		20:	// Close A
      IF TRUE
      AND THIS^.itfValve_LockA.M_ToHP(tDelay:= T#0MS)
			THEN 
        THIS^.stSeqCtrlGeneral.iInternalSeqStateCase := 30;
			END_IF
      
    30:	// Check if open B
      IF TRUE
			THEN 
        IF THIS^.bOpenChB THEN
          THIS^.stSeqCtrlGeneral.iInternalSeqStateCase := 40;
        ELSE
          THIS^.stSeqCtrlGeneral.iInternalSeqStateCase := 50;
        END_IF
			END_IF

    40:	// Open B
      IF TRUE
      AND THIS^.itfValve_LockB.M_ToWP1(tDelay:= T#0MS)
			THEN 
        THIS^.stSeqCtrlGeneral.iInternalSeqStateCase := 1000;
			END_IF
      
		50:	// Close B
      IF TRUE
      AND THIS^.itfValve_LockB.M_ToHP(tDelay:= T#0MS)
			THEN 
        THIS^.stSeqCtrlGeneral.iInternalSeqStateCase := 1000;
			END_IF
      
    1000: // Exit step
      IF TRUE
			THEN 
				THIS^.stSeqCtrlGeneral.iInternalSeqStateCase := 9999;
			END_IF
      
	ELSE
		THIS^.stSeqCtrlGeneral.eActiveSeqState := E_SEQ_GENERAL.DONE;  
	END_CASE
	THIS^.stSeqCtrlGeneral.strExtraInfo := CONCAT('Internal state: ', TO_STRING(THIS^.stSeqCtrlGeneral.iInternalSeqStateCase));

E_SEQ_GENERAL.DONE:;

E_SEQ_GENERAL.ERROR:;

E_SEQ_GENERAL.TIME_OUT:; 
IF TRUE
AND THIS^.stSeqCtrlGeneral.bTimeOutActiveQuit 
THEN
  THIS^.stSeqCtrlGeneral.strExtraInfo := 'Bitte quittieren und erneut testen';
  IF TRUE
  //AND itfOpMode.P_QUIT
  THEN
    THIS^.stSeqCtrlGeneral.eActiveSeqState := E_SEQ_GENERAL.EXECUTE;
	END_IF
  
END_IF

ELSE
  THIS^.stSeqCtrlGeneral.eActiveSeqState := E_SEQ_GENERAL.ERROR;
END_CASE
END_METHOD

METHOD PRIVATE _m_Seq_PRESSURE_CALIBRATION : E_SEQ_PROCESS
VAR_INPUT
END_VAR
VAR
	ActiveSeq:  STRING;
END_VAR
//THIS^._m_GeneralStepSetting(StepType:=E_STEP_STATE_TYPE.INIT,
ActiveSeq := TO_STRING(THIS^.eSeq);

CASE THIS^.stSeqCtrlGeneral.eActiveSeqState OF
E_SEQ_GENERAL.READY:;

	
E_SEQ_GENERAL.EXECUTE:;
	IF TRUE
	THEN
		THIS^.stSeqCtrlGeneral.eActiveSeqState := E_SEQ_GENERAL.RESET;
	END_IF
  
E_SEQ_GENERAL.RESET:;
	stSeqCtrlGeneral.iInternalSeqStateCase := 0;
	IF TRUE
	THEN
    THIS^.ii := 1;
    FOR THIS^.ii := 1 TO 7 BY 1 DO
      THIS^.listCalibrationTable[THIS^.ii].uiValue := 0;
      THIS^.listCalibrationTable[THIS^.ii].uiPressure := 0;
      THIS^.listCalibrationTable[THIS^.ii].uiState := 0;
		END_FOR
    THIS^.ii := 1;
		THIS^.stSeqCtrlGeneral.eActiveSeqState := E_SEQ_GENERAL.BUSY;
	END_IF
  
E_SEQ_GENERAL.BUSY:;
	CASE THIS^.stSeqCtrlGeneral.iInternalSeqStateCase OF
		0:	// Set work pressure value to XXXX
      IF TRUE
      AND THIS^.itfValve_PressureLimit.M_SetLimit(ePressureType:= E_PRESSURE_TYPE.VALUE, rLimit:= 1000 * THIS^.ii)
			THEN 
        THIS^.listCalibrationTable[THIS^.ii].uiValue := TO_UINT(1000 * THIS^.ii);
        THIS^.listCalibrationTable[THIS^.ii].uiState := 1;
        THIS^.stSeqCtrlGeneral.iInternalSeqStateCase := 10;
			END_IF
      
    10:	// Open A channel
      IF TRUE
      AND THIS^.itfValve_LockA.M_ToWP1(tDelay:= T#10MS)
			THEN 
        IF THIS^.bDoableActing THEN
				  THIS^.stSeqCtrlGeneral.iInternalSeqStateCase := 20;
        ELSE
          THIS^.stSeqCtrlGeneral.iInternalSeqStateCase := 30;
        END_IF
			END_IF
      
    20:	// Open B channel
      IF TRUE
      AND THIS^.itfValve_LockB.M_ToWP1(tDelay:= T#10MS)
			THEN 
				THIS^.stSeqCtrlGeneral.iInternalSeqStateCase := 30;
			END_IF
      
    30: // Move cylinder to WP
      IF TRUE
      AND THIS^.itfValve_CylCtrl.M_ValveCtrl(rSpeedInPercent:= 100, tDelay:= T#10MS)
			THEN 
        THIS^.stSeqCtrlGeneral.iInternalSeqStateCase := 40;
			END_IF
      
    40: // Choice step
      IF TRUE
      THEN
        IF THIS^.ii = 1 THEN
          THIS^.stSeqCtrlGeneral.iInternalSeqStateCase := 50;
        ELSE
          THIS^.stSeqCtrlGeneral.iInternalSeqStateCase := 60;
				END_IF
			END_IF
      
    50: // Delay step (wait for cylinder end position)
      IF TRUE
      AND _m_Delay(DelayTime:= T#30S)
      THEN
        THIS^.stSeqCtrlGeneral.iInternalSeqStateCase := 60;
			END_IF
      
    60: // Delay step (cylinder under load)
      IF TRUE
      AND _m_Delay(DelayTime:= T#5S)
      THEN
        THIS^.stSeqCtrlGeneral.iInternalSeqStateCase := 70;
			END_IF
      
    70: // Save pressure
      IF TRUE
      THEN
        THIS^.listCalibrationTable[THIS^.ii].uiPressure := TO_UINT(THIS^.rCurrentPressureInBar);
        THIS^.listCalibrationTable[THIS^.ii].uiState := 2;
        THIS^.stSeqCtrlGeneral.iInternalSeqStateCase := 80;
			END_IF
      
    80: // Decide step
      IF TRUE
      AND _m_Delay(DelayTime:= T#1S)
      THEN
        IF THIS^.ii >= 7 OR THIS^.ii < 1 THEN
          THIS^.ii := 1;
          THIS^.stSeqCtrlGeneral.iInternalSeqStateCase := 1000;
        ELSE
          THIS^.ii := THIS^.ii + 1;
          THIS^.stSeqCtrlGeneral.iInternalSeqStateCase := 0;
				END_IF
			END_IF
      
    1000: // Stop and exit
      IF TRUE
      AND THIS^.itfValve_PressureLimit.M_SetLimit(ePressureType:= E_PRESSURE_TYPE.VALUE, rLimit:= 0)
      AND THIS^.itfValve_CylCtrl.M_ValveCtrl(rSpeedInPercent:= 0, tDelay:= T#10MS)
      AND THIS^.itfValve_LockA.M_ToHP(tDelay:= T#10MS)
      AND THIS^.itfValve_LockB.M_ToHP(tDelay:= T#10MS)
			THEN 
				THIS^.stSeqCtrlGeneral.iInternalSeqStateCase := 9999;
			END_IF
      
	ELSE
		THIS^.stSeqCtrlGeneral.eActiveSeqState := E_SEQ_GENERAL.DONE;  
	END_CASE
	THIS^.stSeqCtrlGeneral.strExtraInfo := CONCAT('Internal state: ', TO_STRING(THIS^.stSeqCtrlGeneral.iInternalSeqStateCase));

E_SEQ_GENERAL.DONE:;

E_SEQ_GENERAL.ERROR:;

E_SEQ_GENERAL.TIME_OUT:; 
IF TRUE
AND THIS^.stSeqCtrlGeneral.bTimeOutActiveQuit 
THEN
  THIS^.stSeqCtrlGeneral.strExtraInfo := 'Bitte quittieren und erneut testen';
  IF TRUE
  //AND itfOpMode.P_QUIT
  THEN
    THIS^.stSeqCtrlGeneral.eActiveSeqState := E_SEQ_GENERAL.EXECUTE;
	END_IF
  
END_IF

ELSE
  THIS^.stSeqCtrlGeneral.eActiveSeqState := E_SEQ_GENERAL.ERROR;
END_CASE
END_METHOD

METHOD PRIVATE _m_Seq_SET_MAX_POS : E_SEQ_PROCESS
VAR_INPUT
END_VAR
VAR
	ActiveSeq: STRING;
END_VAR
VAR
	
END_VAR
//THIS^._m_GeneralStepSetting(StepType:=E_STEP_STATE_TYPE.INIT,
ActiveSeq := TO_STRING(THIS^.eSeq);

CASE THIS^.stSeqCtrlGeneral.eActiveSeqState OF
E_SEQ_GENERAL.READY:;

	
E_SEQ_GENERAL.EXECUTE:;
	IF TRUE
	THEN
		THIS^.stSeqCtrlGeneral.eActiveSeqState := E_SEQ_GENERAL.RESET;
	END_IF
  
E_SEQ_GENERAL.RESET:;
	stSeqCtrlGeneral.iInternalSeqStateCase := 0;
	IF TRUE
	THEN
		THIS^.stSeqCtrlGeneral.eActiveSeqState := E_SEQ_GENERAL.BUSY;
	END_IF
  
E_SEQ_GENERAL.BUSY:;
	CASE THIS^.stSeqCtrlGeneral.iInternalSeqStateCase OF
		0:	// Set max position
      IF TRUE 
			THEN 
        THIS^.lrPosMax := THIS^.lrCurrentPosAbs / 1000;
        THIS^.stSeqCtrlGeneral.iInternalSeqStateCase := 1000;
			END_IF
      
    1000: // Exit step
      IF TRUE
			THEN 
				THIS^.stSeqCtrlGeneral.iInternalSeqStateCase := 9999;
			END_IF
      
	ELSE
		THIS^.stSeqCtrlGeneral.eActiveSeqState := E_SEQ_GENERAL.DONE;  
	END_CASE
	THIS^.stSeqCtrlGeneral.strExtraInfo := CONCAT('Internal state: ', TO_STRING(THIS^.stSeqCtrlGeneral.iInternalSeqStateCase));

E_SEQ_GENERAL.DONE:;

E_SEQ_GENERAL.ERROR:;

E_SEQ_GENERAL.TIME_OUT:; 
IF TRUE
AND THIS^.stSeqCtrlGeneral.bTimeOutActiveQuit 
THEN
  THIS^.stSeqCtrlGeneral.strExtraInfo := 'Bitte quittieren und erneut testen';
  IF TRUE
  //AND itfOpMode.P_QUIT
  THEN
    THIS^.stSeqCtrlGeneral.eActiveSeqState := E_SEQ_GENERAL.EXECUTE;
	END_IF
  
END_IF

ELSE
  THIS^.stSeqCtrlGeneral.eActiveSeqState := E_SEQ_GENERAL.ERROR;
END_CASE
END_METHOD

METHOD PRIVATE _m_Seq_SET_WORK_PRESSURE : E_SEQ_PROCESS
VAR_INPUT
END_VAR
VAR
	ActiveSeq: STRING;
END_VAR
VAR
	
END_VAR
//THIS^._m_GeneralStepSetting(StepType:=E_STEP_STATE_TYPE.INIT,
ActiveSeq := TO_STRING(THIS^.eSeq);

CASE THIS^.stSeqCtrlGeneral.eActiveSeqState OF
E_SEQ_GENERAL.READY:;

	
E_SEQ_GENERAL.EXECUTE:;
	IF TRUE
	THEN
		THIS^.stSeqCtrlGeneral.eActiveSeqState := E_SEQ_GENERAL.RESET;
	END_IF
  
E_SEQ_GENERAL.RESET:;
	stSeqCtrlGeneral.iInternalSeqStateCase := 0;
	IF TRUE
	THEN
		THIS^.stSeqCtrlGeneral.eActiveSeqState := E_SEQ_GENERAL.BUSY;
	END_IF
  
E_SEQ_GENERAL.BUSY:;
	CASE THIS^.stSeqCtrlGeneral.iInternalSeqStateCase OF
		0:	// Set work pressure
      IF TRUE
      AND THIS^.itfValve_PressureLimit.M_SetLimit(ePressureType:= E_PRESSURE_TYPE.VALUE, rLimit:= TO_REAL(THIS^.iTargetPressureAsValueA))
			THEN 
        THIS^.stSeqCtrlGeneral.iInternalSeqStateCase := 1000;
			END_IF
      
    1000: // Exit step
      IF TRUE
			THEN 
				THIS^.stSeqCtrlGeneral.iInternalSeqStateCase := 9999;
			END_IF
      
	ELSE
		THIS^.stSeqCtrlGeneral.eActiveSeqState := E_SEQ_GENERAL.DONE;  
	END_CASE
	THIS^.stSeqCtrlGeneral.strExtraInfo := CONCAT('Internal state: ', TO_STRING(THIS^.stSeqCtrlGeneral.iInternalSeqStateCase));

E_SEQ_GENERAL.DONE:;

E_SEQ_GENERAL.ERROR:;

E_SEQ_GENERAL.TIME_OUT:; 
IF TRUE
AND THIS^.stSeqCtrlGeneral.bTimeOutActiveQuit 
THEN
  THIS^.stSeqCtrlGeneral.strExtraInfo := 'Bitte quittieren und erneut testen';
  IF TRUE
  //AND itfOpMode.P_QUIT
  THEN
    THIS^.stSeqCtrlGeneral.eActiveSeqState := E_SEQ_GENERAL.EXECUTE;
	END_IF
  
END_IF

ELSE
  THIS^.stSeqCtrlGeneral.eActiveSeqState := E_SEQ_GENERAL.ERROR;
END_CASE
END_METHOD

METHOD PRIVATE _m_Seq_SET_WORK_PRESSURE_ZERO : E_SEQ_PROCESS
VAR_INPUT
END_VAR
VAR
	ActiveSeq: STRING;
END_VAR
VAR
	
END_VAR
//THIS^._m_GeneralStepSetting(StepType:=E_STEP_STATE_TYPE.INIT,
ActiveSeq := TO_STRING(THIS^.eSeq);

CASE THIS^.stSeqCtrlGeneral.eActiveSeqState OF
E_SEQ_GENERAL.READY:;

	
E_SEQ_GENERAL.EXECUTE:;
	IF TRUE
	THEN
		THIS^.stSeqCtrlGeneral.eActiveSeqState := E_SEQ_GENERAL.RESET;
	END_IF
  
E_SEQ_GENERAL.RESET:;
	stSeqCtrlGeneral.iInternalSeqStateCase := 0;
	IF TRUE
	THEN
		THIS^.stSeqCtrlGeneral.eActiveSeqState := E_SEQ_GENERAL.BUSY;
	END_IF
  
E_SEQ_GENERAL.BUSY:;
	CASE THIS^.stSeqCtrlGeneral.iInternalSeqStateCase OF
		0:	// Set work pressure
      IF TRUE
      AND THIS^.itfValve_PressureLimit.M_SetLimit(ePressureType:= E_PRESSURE_TYPE.VALUE, rLimit:= 0.0)
			THEN 
        THIS^.stSeqCtrlGeneral.iInternalSeqStateCase := 1000;
			END_IF
      
    1000: // Exit step
      IF TRUE
			THEN 
				THIS^.stSeqCtrlGeneral.iInternalSeqStateCase := 9999;
			END_IF
      
	ELSE
		THIS^.stSeqCtrlGeneral.eActiveSeqState := E_SEQ_GENERAL.DONE;  
	END_CASE
	THIS^.stSeqCtrlGeneral.strExtraInfo := CONCAT('Internal state: ', TO_STRING(THIS^.stSeqCtrlGeneral.iInternalSeqStateCase));

E_SEQ_GENERAL.DONE:;

E_SEQ_GENERAL.ERROR:;

E_SEQ_GENERAL.TIME_OUT:; 
IF TRUE
AND THIS^.stSeqCtrlGeneral.bTimeOutActiveQuit 
THEN
  THIS^.stSeqCtrlGeneral.strExtraInfo := 'Bitte quittieren und erneut testen';
  IF TRUE
  //AND itfOpMode.P_QUIT
  THEN
    THIS^.stSeqCtrlGeneral.eActiveSeqState := E_SEQ_GENERAL.EXECUTE;
	END_IF
  
END_IF

ELSE
  THIS^.stSeqCtrlGeneral.eActiveSeqState := E_SEQ_GENERAL.ERROR;
END_CASE
END_METHOD

METHOD PRIVATE _m_Seq_SET_ZERO_POS : E_SEQ_PROCESS
VAR_INPUT
END_VAR
VAR
	ActiveSeq: STRING;
END_VAR
VAR
	
END_VAR
//THIS^._m_GeneralStepSetting(StepType:=E_STEP_STATE_TYPE.INIT,
ActiveSeq := TO_STRING(THIS^.eSeq);

CASE THIS^.stSeqCtrlGeneral.eActiveSeqState OF
E_SEQ_GENERAL.READY:;

	
E_SEQ_GENERAL.EXECUTE:;
	IF TRUE
	THEN
		THIS^.stSeqCtrlGeneral.eActiveSeqState := E_SEQ_GENERAL.RESET;
	END_IF
  
E_SEQ_GENERAL.RESET:;
	stSeqCtrlGeneral.iInternalSeqStateCase := 0;
	IF TRUE
	THEN
		THIS^.stSeqCtrlGeneral.eActiveSeqState := E_SEQ_GENERAL.BUSY;
	END_IF
  
E_SEQ_GENERAL.BUSY:;
	CASE THIS^.stSeqCtrlGeneral.iInternalSeqStateCase OF
		0:	// Set zero position
      IF TRUE 
			THEN 
        THIS^.lrPosZero := THIS^.lrCurrentPosAbs / 1000;
        THIS^.stSeqCtrlGeneral.iInternalSeqStateCase := 1000;
			END_IF
      
    1000: // Exit step
      IF TRUE
			THEN 
				THIS^.stSeqCtrlGeneral.iInternalSeqStateCase := 9999;
			END_IF
      
	ELSE
		THIS^.stSeqCtrlGeneral.eActiveSeqState := E_SEQ_GENERAL.DONE;  
	END_CASE
	THIS^.stSeqCtrlGeneral.strExtraInfo := CONCAT('Internal state: ', TO_STRING(THIS^.stSeqCtrlGeneral.iInternalSeqStateCase));

E_SEQ_GENERAL.DONE:;

E_SEQ_GENERAL.ERROR:;

E_SEQ_GENERAL.TIME_OUT:; 
IF TRUE
AND THIS^.stSeqCtrlGeneral.bTimeOutActiveQuit 
THEN
  THIS^.stSeqCtrlGeneral.strExtraInfo := 'Bitte quittieren und erneut testen';
  IF TRUE
  //AND itfOpMode.P_QUIT
  THEN
    THIS^.stSeqCtrlGeneral.eActiveSeqState := E_SEQ_GENERAL.EXECUTE;
	END_IF
  
END_IF

ELSE
  THIS^.stSeqCtrlGeneral.eActiveSeqState := E_SEQ_GENERAL.ERROR;
END_CASE
END_METHOD

METHOD PRIVATE _m_Seq_STOP : E_SEQ_PROCESS
VAR_INPUT
END_VAR
VAR
	ActiveSeq: STRING;
END_VAR
VAR
	
END_VAR
//THIS^._m_GeneralStepSetting(StepType:=E_STEP_STATE_TYPE.INIT,
ActiveSeq := TO_STRING(THIS^.eSeq);

CASE THIS^.stSeqCtrlGeneral.eActiveSeqState OF
E_SEQ_GENERAL.READY:;

	
E_SEQ_GENERAL.EXECUTE:;
	IF TRUE
	THEN
    THIS^.bRegulationTrigger := FALSE;
    THIS^.bPressureRegulationTrigger := FALSE;
		THIS^.stSeqCtrlGeneral.eActiveSeqState := E_SEQ_GENERAL.RESET;
	END_IF
  
E_SEQ_GENERAL.RESET:;
	stSeqCtrlGeneral.iInternalSeqStateCase := 0;
	IF TRUE
	THEN
		THIS^.stSeqCtrlGeneral.eActiveSeqState := E_SEQ_GENERAL.BUSY;
	END_IF
  
E_SEQ_GENERAL.BUSY:;
	CASE THIS^.stSeqCtrlGeneral.iInternalSeqStateCase OF
		0: // Switch off valves
      IF TRUE
      AND THIS^.itfValve_CylCtrl.M_ValveCtrl(rSpeedInPercent:= 0, tDelay:= T#0MS)
			THEN 
				THIS^.stSeqCtrlGeneral.iInternalSeqStateCase := 1000;
			END_IF
      
    1000: // Exit step
      IF TRUE
			THEN 
				THIS^.stSeqCtrlGeneral.iInternalSeqStateCase := 9999;
			END_IF
      
	ELSE
		THIS^.stSeqCtrlGeneral.eActiveSeqState := E_SEQ_GENERAL.DONE;  
	END_CASE
	THIS^.stSeqCtrlGeneral.strExtraInfo := CONCAT('Internal state: ', TO_STRING(THIS^.stSeqCtrlGeneral.iInternalSeqStateCase));

E_SEQ_GENERAL.DONE:;

E_SEQ_GENERAL.ERROR:;

E_SEQ_GENERAL.TIME_OUT:; 
IF TRUE
AND THIS^.stSeqCtrlGeneral.bTimeOutActiveQuit 
THEN
  THIS^.stSeqCtrlGeneral.strExtraInfo := 'Bitte quittieren und erneut testen';
  IF TRUE
  //AND itfOpMode.P_QUIT
  THEN
    THIS^.stSeqCtrlGeneral.eActiveSeqState := E_SEQ_GENERAL.EXECUTE;
	END_IF
  
END_IF

ELSE
  THIS^.stSeqCtrlGeneral.eActiveSeqState := E_SEQ_GENERAL.ERROR;
END_CASE
END_METHOD

METHOD PRIVATE _m_Seq_STOP_AND_LOCK : E_SEQ_PROCESS
VAR_INPUT
END_VAR
VAR
	ActiveSeq: STRING;
END_VAR
VAR
	
END_VAR
//THIS^._m_GeneralStepSetting(StepType:=E_STEP_STATE_TYPE.INIT,
ActiveSeq := TO_STRING(THIS^.eSeq);

CASE THIS^.stSeqCtrlGeneral.eActiveSeqState OF
E_SEQ_GENERAL.READY:;

	
E_SEQ_GENERAL.EXECUTE:;
	IF TRUE
	THEN
    THIS^.bRegulationTrigger := FALSE;
    THIS^.bPressureRegulationTrigger := FALSE;
		THIS^.stSeqCtrlGeneral.eActiveSeqState := E_SEQ_GENERAL.RESET;
	END_IF
  
E_SEQ_GENERAL.RESET:;
	stSeqCtrlGeneral.iInternalSeqStateCase := 0;
	IF TRUE
	THEN
		THIS^.stSeqCtrlGeneral.eActiveSeqState := E_SEQ_GENERAL.BUSY;
	END_IF
  
E_SEQ_GENERAL.BUSY:;
	CASE THIS^.stSeqCtrlGeneral.iInternalSeqStateCase OF
		0: // Switch off valves
      IF TRUE
      AND THIS^.itfValve_CylCtrl.M_ValveCtrl(rSpeedInPercent:= 0, tDelay:= T#0MS)
      AND THIS^.itfValve_LockA.M_ToHP(tDelay:= T#0MS)
      AND THIS^.itfValve_LockB.M_ToHP(tDelay:= T#0MS)
			THEN 
				THIS^.stSeqCtrlGeneral.iInternalSeqStateCase := 1000;
			END_IF
      
    1000: // Exit step
      IF TRUE
			THEN 
				THIS^.stSeqCtrlGeneral.iInternalSeqStateCase := 9999;
			END_IF
      
	ELSE
		THIS^.stSeqCtrlGeneral.eActiveSeqState := E_SEQ_GENERAL.DONE;  
	END_CASE
	THIS^.stSeqCtrlGeneral.strExtraInfo := CONCAT('Internal state: ', TO_STRING(THIS^.stSeqCtrlGeneral.iInternalSeqStateCase));

E_SEQ_GENERAL.DONE:;

E_SEQ_GENERAL.ERROR:;

E_SEQ_GENERAL.TIME_OUT:; 
IF TRUE
AND THIS^.stSeqCtrlGeneral.bTimeOutActiveQuit 
THEN
  THIS^.stSeqCtrlGeneral.strExtraInfo := 'Bitte quittieren und erneut testen';
  IF TRUE
  //AND itfOpMode.P_QUIT
  THEN
    THIS^.stSeqCtrlGeneral.eActiveSeqState := E_SEQ_GENERAL.EXECUTE;
	END_IF
  
END_IF

ELSE
  THIS^.stSeqCtrlGeneral.eActiveSeqState := E_SEQ_GENERAL.ERROR;
END_CASE
END_METHOD

METHOD PRIVATE _m_Seq_TO_HP : E_SEQ_PROCESS
VAR_INPUT
END_VAR
VAR
	ActiveSeq: STRING;
END_VAR
//THIS^._m_GeneralStepSetting(StepType:=E_STEP_STATE_TYPE.INIT,
ActiveSeq := TO_STRING(THIS^.eSeq);

CASE THIS^.stSeqCtrlGeneral.eActiveSeqState OF
E_SEQ_GENERAL.READY:;

	
E_SEQ_GENERAL.EXECUTE:;
	IF TRUE
	THEN
    THIS^.bRegulationTrigger := FALSE;
    THIS^.bPressureRegulationTrigger := FALSE;
		THIS^.stSeqCtrlGeneral.eActiveSeqState := E_SEQ_GENERAL.RESET;
	END_IF
  
E_SEQ_GENERAL.RESET:;
	stSeqCtrlGeneral.iInternalSeqStateCase := 0;
	IF TRUE
	THEN
		THIS^.stSeqCtrlGeneral.eActiveSeqState := E_SEQ_GENERAL.BUSY;
	END_IF
  
E_SEQ_GENERAL.BUSY:;
	CASE THIS^.stSeqCtrlGeneral.iInternalSeqStateCase OF
		0:	// Set work pressure
      IF TRUE
      AND THIS^.itfValve_PressureLimit.M_SetLimit(ePressureType:= E_PRESSURE_TYPE.VALUE, rLimit:= TO_REAL(THIS^.iTargetPressureAsValueB))
			THEN 
        THIS^.stSeqCtrlGeneral.iInternalSeqStateCase := 10;
			END_IF
    
    10:	// Switch on lock A valve
      IF TRUE
      AND THIS^.itfValve_LockA.M_ToWP1(tDelay:= T#0MS)
			THEN 
        IF THIS^.bDoableActing THEN
          THIS^.stSeqCtrlGeneral.iInternalSeqStateCase := 20;
        ELSE
          THIS^.stSeqCtrlGeneral.iInternalSeqStateCase := 30;
        END_IF
			END_IF
      
    20:	// Switch on lock B valve
      IF TRUE
      AND THIS^.itfValve_LockB.M_ToWP1(tDelay:= T#0MS)
			THEN 
        THIS^.stSeqCtrlGeneral.iInternalSeqStateCase := 30;
			END_IF
      
    30:	// Set valve control
      IF TRUE
      AND THIS^.itfValve_CylCtrl.M_ValveCtrl(rSpeedInPercent:= THIS^.rSpeedInPercentToSet, tDelay:= T#0MS)
			THEN 
        THIS^.stSeqCtrlGeneral.iInternalSeqStateCase := 1000;
			END_IF
      
    1000: // Exit step
      IF TRUE
			THEN 
				THIS^.stSeqCtrlGeneral.iInternalSeqStateCase := 9999;
			END_IF
      
	ELSE
		THIS^.stSeqCtrlGeneral.eActiveSeqState := E_SEQ_GENERAL.DONE;  
	END_CASE
	THIS^.stSeqCtrlGeneral.strExtraInfo := CONCAT('Internal state: ', TO_STRING(THIS^.stSeqCtrlGeneral.iInternalSeqStateCase));

E_SEQ_GENERAL.DONE:;
  THIS^.bRegulationTrigger := THIS^.bRegulation;
  THIS^.bPressureRegulationTrigger := THIS^.bPressureRegulation;

E_SEQ_GENERAL.ERROR:;

E_SEQ_GENERAL.TIME_OUT:; 
IF TRUE
AND THIS^.stSeqCtrlGeneral.bTimeOutActiveQuit 
THEN
  THIS^.stSeqCtrlGeneral.strExtraInfo := 'Bitte quittieren und erneut testen';
  IF TRUE
  //AND itfOpMode.P_QUIT
  THEN
    THIS^.stSeqCtrlGeneral.eActiveSeqState := E_SEQ_GENERAL.EXECUTE;
	END_IF
  
END_IF

ELSE
  THIS^.stSeqCtrlGeneral.eActiveSeqState := E_SEQ_GENERAL.ERROR;
END_CASE
END_METHOD

METHOD PRIVATE _m_Seq_TO_SET_POS : E_SEQ_PROCESS
VAR_INPUT
END_VAR
VAR
	ActiveSeq: STRING;
END_VAR
VAR
	
END_VAR
//THIS^._m_GeneralStepSetting(StepType:=E_STEP_STATE_TYPE.INIT,
ActiveSeq := TO_STRING(THIS^.eSeq);

CASE THIS^.stSeqCtrlGeneral.eActiveSeqState OF
E_SEQ_GENERAL.READY:;

	
E_SEQ_GENERAL.EXECUTE:;
	IF TRUE
	THEN
		THIS^.stSeqCtrlGeneral.eActiveSeqState := E_SEQ_GENERAL.RESET;
	END_IF
  
E_SEQ_GENERAL.RESET:;
	stSeqCtrlGeneral.iInternalSeqStateCase := 0;
	IF TRUE
	THEN
		THIS^.stSeqCtrlGeneral.eActiveSeqState := E_SEQ_GENERAL.BUSY;
	END_IF
  
E_SEQ_GENERAL.BUSY:;
	CASE THIS^.stSeqCtrlGeneral.iInternalSeqStateCase OF
		0:	// Switch valves
      IF TRUE
      AND THIS^.itfValve_LockA.M_ToWP1(tDelay:= T#10MS)
      AND THIS^.itfValve_LockB.M_ToWP1(tDelay:= T#10MS)
			THEN 
        IF bStrokeLengthInitialized 
        AND THIS^.lrToSetPos <= THIS^.rStrokeLength 
        AND THIS^.lrToSetPos >= 0.0 
        THEN
          // Set direction
          IF THIS^.lrPos > THIS^.lrToSetPos THEN
            THIS^.rSpeedInPercentToSet := -ABS(THIS^.rSpeedInPercentToSet);
			    END_IF
          THIS^.stSeqCtrlGeneral.iInternalSeqStateCase := 10;
        ELSE
          THIS^.stSeqCtrlGeneral.eActiveSeqState := E_SEQ_GENERAL.ERROR;
				END_IF
			END_IF
      
    10: // Move cylinder to HP and wait for endposition
      IF TRUE
      AND THIS^.itfValve_CylCtrl.M_ValveCtrl(rSpeedInPercent:= THIS^.rSpeedInPercentToSet, tDelay:= T#10MS)
			THEN 
        IF THIS^.lrPos < THIS^.rEndPosTol THEN
				  THIS^.stSeqCtrlGeneral.iInternalSeqStateCase := 20;
        END_IF
			END_IF
      
    20: // Switch off valves
      IF TRUE
      AND THIS^.itfValve_CylCtrl.M_ValveCtrl(rSpeedInPercent:= 0, tDelay:= T#10MS)
			THEN 
				THIS^.stSeqCtrlGeneral.iInternalSeqStateCase := 1000;
			END_IF
      
    1000: // Exit step
      IF TRUE
			THEN 
				THIS^.stSeqCtrlGeneral.iInternalSeqStateCase := 9999;
			END_IF
      
	ELSE
		THIS^.stSeqCtrlGeneral.eActiveSeqState := E_SEQ_GENERAL.DONE;  
	END_CASE
	THIS^.stSeqCtrlGeneral.strExtraInfo := CONCAT('Internal state: ', TO_STRING(THIS^.stSeqCtrlGeneral.iInternalSeqStateCase));

E_SEQ_GENERAL.DONE:;

E_SEQ_GENERAL.ERROR:;

E_SEQ_GENERAL.TIME_OUT:; 
IF TRUE
AND THIS^.stSeqCtrlGeneral.bTimeOutActiveQuit 
THEN
  THIS^.stSeqCtrlGeneral.strExtraInfo := 'Bitte quittieren und erneut testen';
  IF TRUE
  //AND itfOpMode.P_QUIT
  THEN
    THIS^.stSeqCtrlGeneral.eActiveSeqState := E_SEQ_GENERAL.EXECUTE;
	END_IF
  
END_IF

ELSE
  THIS^.stSeqCtrlGeneral.eActiveSeqState := E_SEQ_GENERAL.ERROR;
END_CASE
END_METHOD

METHOD PRIVATE _m_Seq_TO_WP : E_SEQ_PROCESS
VAR_INPUT
END_VAR
VAR
	ActiveSeq: STRING;
END_VAR
VAR
	
END_VAR
//THIS^._m_GeneralStepSetting(StepType:=E_STEP_STATE_TYPE.INIT,
ActiveSeq := TO_STRING(THIS^.eSeq);

CASE THIS^.stSeqCtrlGeneral.eActiveSeqState OF
E_SEQ_GENERAL.READY:;

	
E_SEQ_GENERAL.EXECUTE:;
	IF TRUE
	THEN
    THIS^.bRegulationTrigger := FALSE;
    THIS^.bPressureRegulationTrigger := FALSE;
		THIS^.stSeqCtrlGeneral.eActiveSeqState := E_SEQ_GENERAL.RESET;
	END_IF
  
E_SEQ_GENERAL.RESET:;
	stSeqCtrlGeneral.iInternalSeqStateCase := 0;
	IF TRUE
	THEN
		THIS^.stSeqCtrlGeneral.eActiveSeqState := E_SEQ_GENERAL.BUSY;
	END_IF
  
E_SEQ_GENERAL.BUSY:;
	CASE THIS^.stSeqCtrlGeneral.iInternalSeqStateCase OF
		0:	// Set work pressure
      IF TRUE
      AND THIS^.itfValve_PressureLimit.M_SetLimit(ePressureType:= E_PRESSURE_TYPE.VALUE, rLimit:= TO_REAL(THIS^.iTargetPressureAsValueA))
			THEN 
        THIS^.stSeqCtrlGeneral.iInternalSeqStateCase := 10;
			END_IF

    10:	// Switch on lock A valve
      IF TRUE
      AND THIS^.itfValve_LockA.M_ToWP1(tDelay:= T#0MS)
			THEN 
        IF THIS^.bDoableActing THEN
				  THIS^.stSeqCtrlGeneral.iInternalSeqStateCase := 20;
        ELSE
          THIS^.stSeqCtrlGeneral.iInternalSeqStateCase := 30;
        END_IF
			END_IF
      
    20:	// Switch on lock B valve
      IF TRUE
      AND THIS^.itfValve_LockB.M_ToWP1(tDelay:= T#0MS)
			THEN 
				THIS^.stSeqCtrlGeneral.iInternalSeqStateCase := 30;
			END_IF
      
    30:	// Set valve control
      IF TRUE
      AND THIS^.itfValve_CylCtrl.M_ValveCtrl(rSpeedInPercent:= THIS^.rSpeedInPercentToSet, tDelay:= T#0MS)
			THEN 
				THIS^.stSeqCtrlGeneral.iInternalSeqStateCase := 1000;
			END_IF
      
    1000: // Exit step
      IF TRUE
			THEN 
				THIS^.stSeqCtrlGeneral.iInternalSeqStateCase := 9999;
			END_IF
      
	ELSE
		THIS^.stSeqCtrlGeneral.eActiveSeqState := E_SEQ_GENERAL.DONE;  
	END_CASE
	THIS^.stSeqCtrlGeneral.strExtraInfo := CONCAT('Internal state: ', TO_STRING(THIS^.stSeqCtrlGeneral.iInternalSeqStateCase));

E_SEQ_GENERAL.DONE:;
  THIS^.bRegulationTrigger := THIS^.bRegulation;
  THIS^.bPressureRegulationTrigger := THIS^.bPressureRegulation;
  
E_SEQ_GENERAL.ERROR:;

E_SEQ_GENERAL.TIME_OUT:; 
IF TRUE
AND THIS^.stSeqCtrlGeneral.bTimeOutActiveQuit 
THEN
  THIS^.stSeqCtrlGeneral.strExtraInfo := 'Bitte quittieren und erneut testen';
  IF TRUE
  //AND itfOpMode.P_QUIT
  THEN
    THIS^.stSeqCtrlGeneral.eActiveSeqState := E_SEQ_GENERAL.EXECUTE;
	END_IF
  
END_IF

ELSE
  THIS^.stSeqCtrlGeneral.eActiveSeqState := E_SEQ_GENERAL.ERROR;
END_CASE
END_METHOD

METHOD PRIVATE _m_SequenceManager
VAR_INPUT
END_VAR
IF FALSE
//AND THIS^.eActiveSeqState=DONE 
AND eLastSeq<>eSeq
THEN
	IF THIS^.stSeqCtrlGeneral.eActiveSeqState<>E_SEQ_GENERAL.EXECUTE THEN
		THIS^.stSeqCtrlGeneral.eActiveSeqState:=E_SEQ_GENERAL.READY;
	END_IF
END_IF

eSeq := eNextSeq;

//DelayTimer und TimeOut Timer verwalten
stSeqCtrlGeneral.bActiveStep:=	TRUE
				AND eLastSeq					=	eSeq
				AND stSeqCtrlGeneral.eLastActiveSeqState			=	stSeqCtrlGeneral.eActiveSeqState
				AND	stSeqCtrlGeneral.iLastInternalSeqStateCase	=	stSeqCtrlGeneral.iInternalSeqStateCase
				;
			
IF NOT stSeqCtrlGeneral.bActiveStep THEN
	stSeqCtrlGeneral.bDelayActive:=FALSE;
	stSeqCtrlGeneral.bTimeOutActiveQuit:=FALSE;
	stSeqCtrlGeneral.bTimeOutActiveNoQuit:=FALSE;
  THIS^.stSeqCtrlGeneral.strExtraInfo:='';
END_IF

_m_SaveLastStep();
stSeqCtrlGeneral.tonDelay	(IN:=stSeqCtrlGeneral.bActiveStep AND stSeqCtrlGeneral.bDelayActive, 		PT:=stSeqCtrlGeneral.tDelay);
stSeqCtrlGeneral.tonTimeOut	(IN:=stSeqCtrlGeneral.bActiveStep AND (stSeqCtrlGeneral.bTimeOutActiveNoQuit OR stSeqCtrlGeneral.bTimeOutActiveQuit), 	PT:=stSeqCtrlGeneral.tTimeOut);
stSeqCtrlGeneral.tonStepTime	(IN:= stSeqCtrlGeneral.bActiveStep, PT:= T#24H);

IF stSeqCtrlGeneral.tonTimeOut.Q  THEN
	stSeqCtrlGeneral.eActiveSeqState:=E_SEQ_GENERAL.TIME_OUT;
END_IF

IF stSeqCtrlGeneral.iError<>0 THEN
	eSeq:=E_SEQ_CYLINDER.ERROR_SEQ;
END_IF



eLastSeq					:=	eSeq;
stSeqCtrlGeneral.eLastActiveSeqState			:=	stSeqCtrlGeneral.eActiveSeqState;
stSeqCtrlGeneral.iLastInternalSeqStateCase	:=	stSeqCtrlGeneral.iInternalSeqStateCase;

// Reset set ready state
IF THIS^.stSeqCtrlGeneral.bExitSetReadyState THEN
  THIS^.stSeqCtrlGeneral.bExitSetReadyState := FALSE;
END_IF
END_METHOD

(******************Description****************)
// This function allows variable speed control
(*********************************************)
METHOD PRIVATE _m_SpeedRegulation : BOOL
VAR_INPUT
END_VAR
IF TRUE
AND THIS^.rCurrentSpeedInMmPerS < THIS^.rSpeedInMmPerSToSet 
AND THIS^.rCorrectedSpeedPercent < 100
AND THIS^.bRegulationTrigger
AND NOT THIS^.bRegulationBusy
THEN
  IF ABS(THIS^.rCurrentSpeedInMmPerS - THIS^.rSpeedInMmPerSToSet) > 1 THEN
    //THIS^.rCorrectedSpeedPercent := THIS^.rCorrectedSpeedPercent + 0.25;
    THIS^.rCorrectedSpeedPercent := THIS^.rCorrectedSpeedPercent + ABS((THIS^.rCurrentSpeedInMmPerS - THIS^.rSpeedInMmPerSToSet) * THIS^.rSpeedRegulationFactor);
    THIS^.bCorrectionTrigger := TRUE;
  END_IF
ELSIF TRUE
AND THIS^.rCurrentSpeedInMmPerS > THIS^.rSpeedInMmPerSToSet 
AND THIS^.rCorrectedSpeedPercent > -100
AND THIS^.bRegulationTrigger
AND NOT THIS^.bRegulationBusy
THEN
  IF ABS(THIS^.rCurrentSpeedInMmPerS - THIS^.rSpeedInMmPerSToSet) > 1 THEN
    //THIS^.rCorrectedSpeedPercent := THIS^.rCorrectedSpeedPercent - 0.25;
    THIS^.rCorrectedSpeedPercent := THIS^.rCorrectedSpeedPercent - ABS((THIS^.rCurrentSpeedInMmPerS - THIS^.rSpeedInMmPerSToSet) * THIS^.rSpeedRegulationFactor);
    THIS^.bCorrectionTrigger := TRUE;
  END_IF
END_IF

// Valve value correction
IF THIS^.bCorrectionTrigger THEN
  THIS^.bRegulationBusy:= TRUE;
  CASE THIS^.uiRegulationSeq OF
    0:;
      IF THIS^.itfValve_CylCtrl.M_SetReady() THEN
        THIS^.uiRegulationSeq := 1;
	    END_IF
    1:;
      IF THIS^.itfValve_CylCtrl.M_ValveCtrl(rSpeedInPercent:= THIS^.rCorrectedSpeedPercent, tDelay:= T#0MS) THEN
        THIS^.bCorrectionTrigger := FALSE;
        THIS^.bRegulationBusy := FALSE;
        THIS^.uiRegulationSeq := 0;
	    END_IF
	END_CASE
END_IF
END_METHOD

METHOD PRIVATE _m_TimeOut : BOOL
VAR_INPUT
	bTimeoutActiveToQuit:	BOOL;
	bTimeOutActiveNoQuit:	BOOL;
	tTimeOut:				TIME;	
END_VAR
THIS^.stSeqCtrlGeneral.bTimeOutActiveQuit:=	bTimeoutActiveToQuit;
THIS^.stSeqCtrlGeneral.bTimeOutActiveNoQuit:=	bTimeOutActiveNoQuit;
THIS^.stSeqCtrlGeneral.tTimeOut:=			tTimeOut;
_m_TimeOut:=FALSE;
IF THIS^.stSeqCtrlGeneral.tonTimeOut.Q THEN
	_m_TimeOut:=TRUE;
END_IF
END_METHOD

METHOD FB_init : BOOL
VAR_INPUT
	bInitRetains : BOOL; // if TRUE, the retain variables are initialized (warm start / cold start)
	bInCopyCode : BOOL;  // if TRUE, the instance afterwards gets moved into the copy code (online change)
  
  itfOpMode:											                        I_OP_MODE;
  itfEventLogger:                                         I_EVENT_LOGGER;
  itfOpModeVisu:											                    I_OP_MODE_PAUSE_VISU;
  itfValve_CylCtrl:                                       I_VALVE_X_3_PROP;
  itfValve_LockA:                                         I_VALVE_X_2;
  itfValve_LockB:                                         I_VALVE_X_2;
  itfValve_PressureLimit:                                 I_PRV_PROP; 
  rEndPosTol:                                             REAL;
  /// Volume flow in l/min or dm³/min
  rPumpVolumeFlow:                                        REAL; // Volumenstrom
  /// Pump efficiency factor (0,5-1)
  rPumpEfficiencyFactor:                                  REAL; // Wirkungsgrad
END_VAR
THIS^.itfOpMode := itfOpMode;
THIS^.itfEventLogger := itfEventLogger;
THIS^.itfOpModeVisu := itfOpModeVisu;
THIS^.itfValve_CylCtrl := itfValve_CylCtrl;
THIS^.itfValve_LockA := itfValve_LockA;
THIS^.itfValve_LockB := itfValve_LockB;
THIS^.itfValve_PressureLimit := itfValve_PressureLimit;
THIS^.rEndPosTol := rEndPosTol;
THIS^.rPumpVolumeFlow := rPumpVolumeFlow;
THIS^.rPumpEfficiencyFactor := rPumpEfficiencyFactor;
END_METHOD

METHOD M_OpenLockValves : BOOL
VAR_INPUT
	bOpenChA	: BOOL;
	bOpenChB	: BOOL;
END_VAR
M_OpenLockValves := THIS^.stSeqCtrlGeneral.eActiveSeqState = E_SEQ_GENERAL.DONE;

// Assign input
THIS^.bOpenChA := bOpenChA;
THIS^.bOpenChB := bOpenChB;

// General
IF THIS^.stSeqCtrlGeneral.eActiveSeqState = E_SEQ_GENERAL.READY THEN
  THIS^.eNextSeq := E_SEQ_CYLINDER.OPEN_LOCK_VALVES;
  THIS^.stSeqCtrlGeneral.eActiveSeqState := E_SEQ_GENERAL.EXECUTE;
END_IF
END_METHOD

METHOD M_PressureCalibration : BOOL
M_PressureCalibration := THIS^.stSeqCtrlGeneral.eActiveSeqState = E_SEQ_GENERAL.DONE;

// Assign input

// General
IF THIS^.stSeqCtrlGeneral.eActiveSeqState = E_SEQ_GENERAL.READY THEN
  THIS^.eNextSeq := E_SEQ_CYLINDER.PRESSURE_CALIBRATION;
  THIS^.stSeqCtrlGeneral.eActiveSeqState := E_SEQ_GENERAL.EXECUTE;
END_IF
END_METHOD

METHOD M_Reset : BOOL
M_Reset := THIS^.stSeqCtrlGeneral.eActiveSeqState = E_SEQ_GENERAL.DONE;

// General
IF THIS^.stSeqCtrlGeneral.eActiveSeqState = E_SEQ_GENERAL.READY THEN
  THIS^.eNextSeq := E_SEQ_CYLINDER.INIT;
  THIS^.stSeqCtrlGeneral.eActiveSeqState := E_SEQ_GENERAL.EXECUTE;
END_IF
END_METHOD

{warning 'Methodenimplementierung hinzufügen'}
(*=== Method: M_Run  ============================================

 @brief: Here is the global code (Timer, Event, Flange,...)*)
METHOD M_Run
END_METHOD

METHOD M_SetMaxPos : BOOL
M_SetMaxPos := THIS^.stSeqCtrlGeneral.eActiveSeqState = E_SEQ_GENERAL.DONE;

// General
IF THIS^.stSeqCtrlGeneral.eActiveSeqState = E_SEQ_GENERAL.READY THEN
  THIS^.eNextSeq := E_SEQ_CYLINDER.SET_MAX_POS;
  THIS^.stSeqCtrlGeneral.eActiveSeqState := E_SEQ_GENERAL.EXECUTE;
END_IF
END_METHOD

METHOD M_SetReady : BOOL
VAR_INPUT
END_VAR
M_SetReady := TRUE
              AND THIS^.stSeqCtrlGeneral.eActiveSeqState = E_SEQ_GENERAL.READY
              AND THIS^.eSeq = E_SEQ_CYLINDER.BASE;

THIS^.stSeqCtrlGeneral.eActiveSeqState := E_SEQ_GENERAL.READY;
THIS^.eNextSeq := E_SEQ_CYLINDER.BASE;
END_METHOD

METHOD M_SetWorkPressure : BOOL
VAR_INPUT
  ePressureType:                   E_PRESSURE_TYPE;
  rWorkPressure:                   REAL;
END_VAR
M_SetWorkPressure := THIS^.stSeqCtrlGeneral.eActiveSeqState = E_SEQ_GENERAL.DONE;

// Assign input
IF ePressureType = E_PRESSURE_TYPE.BAR THEN
  THIS^.rTargetPressureInBarA := THIS^.rTargetPressureInBarB := rWorkPressure;
  THIS^.rTargetPressureInForceA := rWorkPressure / 10 * THIS^.lrPistonSurfaceA;
  THIS^.rTargetPressureInForceB := rWorkPressure / 10 * THIS^.lrPistonSurfaceB;
  THIS^.rTargetPressureInPercentA := THIS^.rTargetPressureInPercentB := 100 / THIS^.itfValve_PressureLimit.P_MaxLimitInBar * rWorkPressure;
  THIS^.iTargetPressureAsValueA := THIS^.iTargetPressureAsValueB := TO_INT(F_InterpolLinear(lrValueUnscale := rWorkPressure , arrCalibrate:= listCylCalibration, iPts:= 7));
ELSIF ePressureType = E_PRESSURE_TYPE.FORCE THEN
  THIS^.rTargetPressureInForceA := THIS^.rTargetPressureInForceB := rWorkPressure;;
  THIS^.rTargetPressureInBarA := THIS^.rTargetPressureInForceA / THIS^.lrPistonSurfaceA * 10;
  THIS^.rTargetPressureInBarB := THIS^.rTargetPressureInForceB / THIS^.lrPistonSurfaceB * 10;
  THIS^.rTargetPressureInPercentA := 100 / THIS^.itfValve_PressureLimit.P_MaxLimitInBar * THIS^.rTargetPressureInBarA;
  THIS^.rTargetPressureInPercentB := 100 / THIS^.itfValve_PressureLimit.P_MaxLimitInBar * THIS^.rTargetPressureInBarB;
  THIS^.iTargetPressureAsValueA := TO_INT(F_InterpolLinear(lrValueUnscale := THIS^.rTargetPressureInBarA , arrCalibrate:= listCylCalibration, iPts:= 7));
  THIS^.iTargetPressureAsValueB := TO_INT(F_InterpolLinear(lrValueUnscale := THIS^.rTargetPressureInBarB , arrCalibrate:= listCylCalibration, iPts:= 7));
ELSIF ePressureType = E_PRESSURE_TYPE.PERCENT THEN
  THIS^.rTargetPressureInPercentA := THIS^.rTargetPressureInPercentB := rWorkPressure;
  THIS^.rTargetPressureInBarA := THIS^.rTargetPressureInBarB := THIS^.itfValve_PressureLimit.P_MaxLimitInBar / 100 * rWorkPressure;
  THIS^.rTargetPressureInForceA := THIS^.rTargetPressureInBarA / 10 * THIS^.lrPistonSurfaceA;
  THIS^.rTargetPressureInForceB := THIS^.rTargetPressureInBarB / 10 * THIS^.lrPistonSurfaceB;
  THIS^.iTargetPressureAsValueA := TO_INT(F_InterpolLinear(lrValueUnscale := THIS^.rTargetPressureInBarA , arrCalibrate:= listCylCalibration, iPts:= 7));
  THIS^.iTargetPressureAsValueB := TO_INT(F_InterpolLinear(lrValueUnscale := THIS^.rTargetPressureInBarB , arrCalibrate:= listCylCalibration, iPts:= 7));
ELSE
  THIS^.iTargetPressureAsValueA := THIS^.iTargetPressureAsValueB := TO_INT(rWorkPressure);
END_IF

// General
IF THIS^.stSeqCtrlGeneral.eActiveSeqState = E_SEQ_GENERAL.READY THEN
  THIS^.eNextSeq := E_SEQ_CYLINDER.SET_WORK_PRESSURE;
  THIS^.stSeqCtrlGeneral.eActiveSeqState := E_SEQ_GENERAL.EXECUTE;
END_IF
END_METHOD

METHOD M_SetWorkPressureZero : BOOL
M_SetWorkPressureZero := THIS^.stSeqCtrlGeneral.eActiveSeqState = E_SEQ_GENERAL.DONE;

THIS^.bRegulation := FALSE;
THIS^.rSpeedInMmPerSToSet := 0;
THIS^.rSpeedInPercentToSet := 0;
THIS^.rCorrectedSpeedPercent := 0;
THIS^.bPressureRegulation := FALSE;
THIS^.rActiveForce := 0;
THIS^.iCorrectedPressureAsValue := 0;
THIS^.bPressureRegulationTrigger := FALSE;
THIS^.bPressureRegulationBusy := FALSE;
THIS^.bPressureCorrectionTrigger := FALSE;
THIS^.iTargetPressureAsValueA := 0;

// General
IF THIS^.stSeqCtrlGeneral.eActiveSeqState = E_SEQ_GENERAL.READY THEN
  THIS^.eNextSeq := E_SEQ_CYLINDER.SET_WORK_PRESSURE_ZERO;
  THIS^.stSeqCtrlGeneral.eActiveSeqState := E_SEQ_GENERAL.EXECUTE;
END_IF
END_METHOD

METHOD M_SetZeroPos : BOOL
M_SetZeroPos := THIS^.stSeqCtrlGeneral.eActiveSeqState = E_SEQ_GENERAL.DONE;

// General
IF THIS^.stSeqCtrlGeneral.eActiveSeqState = E_SEQ_GENERAL.READY THEN
  THIS^.eNextSeq := E_SEQ_CYLINDER.SET_ZERO_POS;
  THIS^.stSeqCtrlGeneral.eActiveSeqState := E_SEQ_GENERAL.EXECUTE;
END_IF
END_METHOD

METHOD M_Stop : BOOL
M_Stop := THIS^.stSeqCtrlGeneral.eActiveSeqState = E_SEQ_GENERAL.DONE;

// Assign input
THIS^.bRegulation := FALSE;
THIS^.rSpeedInMmPerSToSet := 0;
THIS^.rSpeedInPercentToSet := 0;
THIS^.rCorrectedSpeedPercent := 0;
THIS^.bPressureRegulation := FALSE;
THIS^.rActiveForce := 0;
THIS^.iCorrectedPressureAsValue := 0;
THIS^.bPressureRegulationTrigger := FALSE;
THIS^.bPressureRegulationBusy := FALSE;
THIS^.bPressureCorrectionTrigger := FALSE;

// General
IF THIS^.stSeqCtrlGeneral.eActiveSeqState = E_SEQ_GENERAL.READY THEN
  THIS^.eNextSeq := E_SEQ_CYLINDER.STOP;
  THIS^.stSeqCtrlGeneral.eActiveSeqState := E_SEQ_GENERAL.EXECUTE;
END_IF
END_METHOD

METHOD M_StopAndLock : BOOL
M_StopAndLock := THIS^.stSeqCtrlGeneral.eActiveSeqState = E_SEQ_GENERAL.DONE;

// Assign input
THIS^.bRegulation := FALSE;
THIS^.rSpeedInMmPerSToSet := 0;
THIS^.rSpeedInPercentToSet := 0;
THIS^.rCorrectedSpeedPercent := 0;
THIS^.bPressureRegulation := FALSE;
THIS^.rActiveForce := 0;
THIS^.iCorrectedPressureAsValue := 0;
THIS^.bPressureRegulationTrigger := FALSE;
THIS^.bPressureRegulationBusy := FALSE;
THIS^.bPressureCorrectionTrigger := FALSE;

// General
IF THIS^.stSeqCtrlGeneral.eActiveSeqState = E_SEQ_GENERAL.READY THEN
  THIS^.eNextSeq := E_SEQ_CYLINDER.STOP_AND_LOCK;
  THIS^.stSeqCtrlGeneral.eActiveSeqState := E_SEQ_GENERAL.EXECUTE;
END_IF
END_METHOD

METHOD M_ToHP : BOOL
VAR_INPUT
  /// Bar | Force in N | Percent 0-100 | Value 0-32767
  ePressureType:            E_PRESSURE_TYPE;
  rWorkPressure:            REAL;
  bPressureRegulation:      BOOL;
  /// Just need for prop valve
  eSpeedType:               E_SPEED_TYPE;
  rSpeed:                   REAL;
END_VAR
VAR
  
END_VAR
M_ToHP := THIS^.stSeqCtrlGeneral.eActiveSeqState = E_SEQ_GENERAL.DONE;

// Der prozentualler Wert wurde pauschal um -15 verringert, da sonst die automatische Regullierung zuviel nachregeln muss (Toter Ventilbereich).
// Hier mit weiteren Varianten testen, wie sich die Regelung verhällt, evtl parametrierbar.

// Assign input
IF eSpeedType = E_SPEED_TYPE.MM_PER_SECOND THEN
  THIS^.bRegulation := TRUE;
  THIS^.rSpeedInMmPerSToSet := -ABS(rSpeed);
  THIS^.rSpeedInPercentToSet := THIS^.rCorrectedSpeedPercent := -15(*-ABS((3 * THIS^.lrPistonSurfaceB * THIS^.rPumpEfficiencyFactor * rSpeed) / (500 * THIS^.rPumpVolumeFlow))*);
ELSE
  THIS^.bRegulation := FALSE;
  THIS^.rSpeedInPercentToSet := THIS^.rCorrectedSpeedPercent := -ABS(rSpeed);
END_IF
IF THIS^.rSpeedInPercentToSet < -100 THEN
  THIS^.rSpeedInPercentToSet := THIS^.rCorrectedSpeedPercent := -100;
END_IF

IF ePressureType = E_PRESSURE_TYPE.BAR THEN
  THIS^.rTargetPressureInBarA := THIS^.rTargetPressureInBarB := rWorkPressure;
  THIS^.rTargetPressureInForceA := rWorkPressure / 10 * THIS^.lrPistonSurfaceA;
  THIS^.rTargetPressureInForceB := rWorkPressure / 10 * THIS^.lrPistonSurfaceB;
  THIS^.rTargetPressureInPercentA := THIS^.rTargetPressureInPercentB := 100 / THIS^.itfValve_PressureLimit.P_MaxLimitInBar * rWorkPressure;
  THIS^.iTargetPressureAsValueA := THIS^.iTargetPressureAsValueB := THIS^.iCorrectedPressureAsValue := TO_INT(F_InterpolLinear(lrValueUnscale := rWorkPressure , arrCalibrate:= listCylCalibration, iPts:= 7));
ELSIF ePressureType = E_PRESSURE_TYPE.FORCE THEN
  THIS^.rTargetPressureInForceA := THIS^.rTargetPressureInForceB := rWorkPressure;;
  THIS^.rTargetPressureInBarA := THIS^.rTargetPressureInForceA / THIS^.lrPistonSurfaceA * 10;
  THIS^.rTargetPressureInBarB := THIS^.rTargetPressureInForceB / THIS^.lrPistonSurfaceB * 10;
  THIS^.rTargetPressureInPercentA := 100 / THIS^.itfValve_PressureLimit.P_MaxLimitInBar * THIS^.rTargetPressureInBarA;
  THIS^.rTargetPressureInPercentB := 100 / THIS^.itfValve_PressureLimit.P_MaxLimitInBar * THIS^.rTargetPressureInBarB;
  THIS^.iTargetPressureAsValueA := THIS^.iCorrectedPressureAsValue := TO_INT(F_InterpolLinear(lrValueUnscale := THIS^.rTargetPressureInBarA , arrCalibrate:= listCylCalibration, iPts:= 7));
  THIS^.iTargetPressureAsValueB := TO_INT(F_InterpolLinear(lrValueUnscale := THIS^.rTargetPressureInBarB , arrCalibrate:= listCylCalibration, iPts:= 7));
ELSIF ePressureType = E_PRESSURE_TYPE.PERCENT THEN
  THIS^.rTargetPressureInPercentA := THIS^.rTargetPressureInPercentB := rWorkPressure;
  THIS^.rTargetPressureInBarA := THIS^.rTargetPressureInBarB := THIS^.itfValve_PressureLimit.P_MaxLimitInBar / 100 * rWorkPressure;
  THIS^.rTargetPressureInForceA := THIS^.rTargetPressureInBarA / 10 * THIS^.lrPistonSurfaceA;
  THIS^.rTargetPressureInForceB := THIS^.rTargetPressureInBarB / 10 * THIS^.lrPistonSurfaceB;
  THIS^.iTargetPressureAsValueA := THIS^.iCorrectedPressureAsValue := TO_INT(F_InterpolLinear(lrValueUnscale := THIS^.rTargetPressureInBarA , arrCalibrate:= listCylCalibration, iPts:= 7));
  THIS^.iTargetPressureAsValueB := TO_INT(F_InterpolLinear(lrValueUnscale := THIS^.rTargetPressureInBarB , arrCalibrate:= listCylCalibration, iPts:= 7));
ELSE
  THIS^.iTargetPressureAsValueA := THIS^.iTargetPressureAsValueB := THIS^.iCorrectedPressureAsValue := TO_INT(rWorkPressure);
END_IF
THIS^.bPressureRegulation := bPressureRegulation;

// General
IF THIS^.stSeqCtrlGeneral.eActiveSeqState = E_SEQ_GENERAL.READY THEN
  THIS^.eNextSeq := E_SEQ_CYLINDER.TO_HP;
  THIS^.stSeqCtrlGeneral.eActiveSeqState := E_SEQ_GENERAL.EXECUTE;
END_IF
END_METHOD

METHOD M_ToSetPos : BOOL
VAR_INPUT
  lrToSetPos:                 LREAL;
  /// Just need for prop valve
  eSpeedType:               E_SPEED_TYPE;
  rSpeed:                   REAL; 
END_VAR
VAR
  lrCylPistonSurface:       LREAL;
END_VAR
M_ToSetPos := THIS^.stSeqCtrlGeneral.eActiveSeqState = E_SEQ_GENERAL.DONE;

// Assign input
THIS^.lrToSetPos := lrToSetPos;
IF eSpeedType = E_SPEED_TYPE.MM_PER_SECOND THEN
  THIS^.rSpeedInMmPerSToSet := rSpeed;
  // Convert mm/s to percent
  IF THIS^.lrPos < lrToSetPos THEN
    lrCylPistonSurface := THIS^.lrPistonSurfaceA;
  ELSE
    lrCylPistonSurface := THIS^.lrPistonSurfaceB;
  END_IF
  THIS^.rSpeedInPercentToSet := ABS((3 * lrCylPistonSurface * THIS^.rPumpEfficiencyFactor * rSpeed) / (500 * THIS^.rPumpVolumeFlow));
ELSE
  THIS^.rSpeedInPercentToSet := ABS(rSpeed);
END_IF
IF THIS^.rSpeedInPercentToSet > 100 THEN
  THIS^.rSpeedInPercentToSet := 100;
END_IF

// General
IF THIS^.stSeqCtrlGeneral.eActiveSeqState = E_SEQ_GENERAL.READY THEN
  THIS^.eNextSeq := E_SEQ_CYLINDER.TO_SET_POS;
  THIS^.stSeqCtrlGeneral.eActiveSeqState := E_SEQ_GENERAL.EXECUTE;
END_IF
END_METHOD

METHOD M_ToWP : BOOL
VAR_INPUT
  /// Bar | Force in N | Percent 0-100 | Value 0-32767
  ePressureType:            E_PRESSURE_TYPE;
  rWorkPressure:            REAL;
  bPressureRegulation:      BOOL;
  /// Just need for prop valve
  eSpeedType:               E_SPEED_TYPE;
  rSpeed:                   REAL;
END_VAR
M_ToWP := THIS^.stSeqCtrlGeneral.eActiveSeqState = E_SEQ_GENERAL.DONE;

// Der prozentualler Wert wurde pauschal um -5 verringert, da sonst die automatische Regullierung zuviel nachregeln muss (Toter Ventilbereich).
// Hier mit weiteren Varianten testen, wie sich die Regelung verhällt, evtl parametrierbar.

// Assign input
IF eSpeedType = E_SPEED_TYPE.MM_PER_SECOND THEN
  THIS^.bRegulation := TRUE;
  THIS^.rSpeedInMmPerSToSet := ABS(rSpeed);
  THIS^.rSpeedInPercentToSet := THIS^.rCorrectedSpeedPercent := 15(*ABS((3 * THIS^.lrPistonSurfaceA * THIS^.rPumpEfficiencyFactor * rSpeed) / (500 * THIS^.rPumpVolumeFlow))*);
ELSE
  THIS^.bRegulation := FALSE;
  THIS^.rSpeedInPercentToSet := THIS^.rCorrectedSpeedPercent := ABS(rSpeed);
END_IF
IF THIS^.rSpeedInPercentToSet > 100 THEN
  THIS^.rSpeedInPercentToSet := THIS^.rCorrectedSpeedPercent := 100;
END_IF

IF ePressureType = E_PRESSURE_TYPE.BAR THEN
  THIS^.rTargetPressureInBarA := THIS^.rTargetPressureInBarB := rWorkPressure;
  THIS^.rTargetPressureInForceA := rWorkPressure / 10 * THIS^.lrPistonSurfaceA;
  THIS^.rTargetPressureInForceB := rWorkPressure / 10 * THIS^.lrPistonSurfaceB;
  THIS^.rTargetPressureInPercentA := THIS^.rTargetPressureInPercentB := 100 / THIS^.itfValve_PressureLimit.P_MaxLimitInBar * rWorkPressure;
  THIS^.iTargetPressureAsValueA := THIS^.iTargetPressureAsValueB := THIS^.iCorrectedPressureAsValue := TO_INT(F_InterpolLinear(lrValueUnscale := rWorkPressure , arrCalibrate:= listCylCalibration, iPts:= 7));
ELSIF ePressureType = E_PRESSURE_TYPE.FORCE THEN
  THIS^.rTargetPressureInForceA := THIS^.rTargetPressureInForceB := rWorkPressure;;
  THIS^.rTargetPressureInBarA := THIS^.rTargetPressureInForceA / THIS^.lrPistonSurfaceA * 10;
  THIS^.rTargetPressureInBarB := THIS^.rTargetPressureInForceB / THIS^.lrPistonSurfaceB * 10;
  THIS^.rTargetPressureInPercentA := 100 / THIS^.itfValve_PressureLimit.P_MaxLimitInBar * THIS^.rTargetPressureInBarA;
  THIS^.rTargetPressureInPercentB := 100 / THIS^.itfValve_PressureLimit.P_MaxLimitInBar * THIS^.rTargetPressureInBarB;
  THIS^.iTargetPressureAsValueA := THIS^.iCorrectedPressureAsValue := TO_INT(F_InterpolLinear(lrValueUnscale := THIS^.rTargetPressureInBarA , arrCalibrate:= listCylCalibration, iPts:= 7));
  THIS^.iTargetPressureAsValueB := TO_INT(F_InterpolLinear(lrValueUnscale := THIS^.rTargetPressureInBarB , arrCalibrate:= listCylCalibration, iPts:= 7));
ELSIF ePressureType = E_PRESSURE_TYPE.PERCENT THEN
  THIS^.rTargetPressureInPercentA := THIS^.rTargetPressureInPercentB := rWorkPressure;
  THIS^.rTargetPressureInBarA := THIS^.rTargetPressureInBarB := THIS^.itfValve_PressureLimit.P_MaxLimitInBar / 100 * rWorkPressure;
  THIS^.rTargetPressureInForceA := THIS^.rTargetPressureInBarA / 10 * THIS^.lrPistonSurfaceA;
  THIS^.rTargetPressureInForceB := THIS^.rTargetPressureInBarB / 10 * THIS^.lrPistonSurfaceB;
  THIS^.iTargetPressureAsValueA := THIS^.iCorrectedPressureAsValue := TO_INT(F_InterpolLinear(lrValueUnscale := THIS^.rTargetPressureInBarA , arrCalibrate:= listCylCalibration, iPts:= 7));
  THIS^.iTargetPressureAsValueB := TO_INT(F_InterpolLinear(lrValueUnscale := THIS^.rTargetPressureInBarB , arrCalibrate:= listCylCalibration, iPts:= 7));
ELSE
  THIS^.iTargetPressureAsValueA := THIS^.iTargetPressureAsValueB := THIS^.iCorrectedPressureAsValue := TO_INT(rWorkPressure);
END_IF
THIS^.bPressureRegulation := bPressureRegulation;

// General
IF THIS^.stSeqCtrlGeneral.eActiveSeqState = E_SEQ_GENERAL.READY THEN
  THIS^.eNextSeq := E_SEQ_CYLINDER.TO_WP;
  THIS^.stSeqCtrlGeneral.eActiveSeqState := E_SEQ_GENERAL.EXECUTE;
END_IF
END_METHOD

PROPERTY P_ActiveDirection : SINT
GET
IF THIS^.itfValve_CylCtrl.P_CurrentVal < - 100 THEN
  P_ActiveDirection := -1;
ELSIF THIS^.itfValve_CylCtrl.P_CurrentVal > 100 THEN
  P_ActiveDirection := 1;
ELSE
  P_ActiveDirection := 0;
END_IF
END_GET
END_PROPERTY

PROPERTY P_CurrentForceInKN : REAL
GET
IF THIS^.rCorrectedSpeedPercent > 0 THEN
  P_CurrentForceInKN := THIS^.rCurrentPressureInBar / 10000 * THIS^.lrPistonSurfaceA;
  THIS^.rActiveForce := THIS^.rTargetPressureInForceA;
ELSE
  P_CurrentForceInKN := THIS^.rCurrentPressureInBar / 10000 * THIS^.lrPistonSurfaceB;
  THIS^.rActiveForce := THIS^.rTargetPressureInForceB;
END_IF
END_GET
END_PROPERTY

{warning 'Eigenschaftenimplementierung hinzufügen'}
PROPERTY P_DoubleActing : BOOL
GET
P_DoubleActing := THIS^.bDoableActing;
END_GET
END_PROPERTY

{warning 'Eigenschaftenimplementierung hinzufügen'}
(*=== Property: P_Event  ============================================

 @param [set]: 	Set the Structure "ST_EVENT" from another Object
 @param [get]: 	Return the Structure "ST_EVENT", it contains the actual 
					event of the Object *)
PROPERTY P_Event : GenLib.ST_EVENT
GET
END_GET
SET
END_SET
END_PROPERTY

{warning 'Eigenschaftenimplementierung hinzufügen'}
(*=== Property: P_FullObjectPath  ============================================

 @param [set]: 	Set the Object Path (Clear String of Object)
 @param [get]: 	Return the Objectpath *)
PROPERTY P_FullObjectPath : STRING
GET
P_FullObjectPath := strInstancePath;
END_GET
SET
strInstancePath := P_FullObjectPath;
END_SET
END_PROPERTY

{warning 'Eigenschaftenimplementierung hinzufügen'}
(*=== Property: P_Global_Ack  ============================================

 @param [set]: 	Set the Bit for Ack from another Object
 @param [get]: 	Return the state of Ack Bit*)
PROPERTY P_Global_Ack : BOOL
GET
END_GET
SET
END_SET
END_PROPERTY

{warning 'Eigenschaftenimplementierung hinzufügen'}
(*=== Property: P_GlobalID  ============================================

 @param [set]: 	-
 @param [get]: 	Return the string of instance path*)
PROPERTY P_GlobalID : STRING
GET
END_GET
END_PROPERTY

{warning 'Eigenschaftenimplementierung hinzufügen'}
PROPERTY P_MaxPosVal : LREAL
GET
P_MaxPosVal := THIS^.lrPosMax;
END_GET
END_PROPERTY

{warning 'Eigenschaftenimplementierung hinzufügen'}
PROPERTY P_MinPosVal : LREAL
GET
P_MinPosVal := THIS^.lrPosZero;
END_GET
END_PROPERTY

{warning 'Eigenschaftenimplementierung hinzufügen'}
PROPERTY P_PistonSurfaceA : LREAL
GET
P_PistonSurfaceA := THIS^.lrPistonSurfaceA;
END_GET
END_PROPERTY

{warning 'Eigenschaftenimplementierung hinzufügen'}
PROPERTY P_PistonSurfaceB : LREAL
GET
P_PistonSurfaceB := THIS^.lrPistonSurfaceB;
END_GET
END_PROPERTY

PROPERTY P_Position : LREAL
GET
P_Position := THIS^.lrPos;
END_GET
END_PROPERTY

{warning 'Eigenschaftenimplementierung hinzufügen'}
PROPERTY P_PositionAbs : LREAL
GET
P_PositionAbs := THIS^.lrCurrentPosAbs / 1000;
END_GET
END_PROPERTY

{warning 'Eigenschaftenimplementierung hinzufügen'}
PROPERTY P_PressureChA : REAL
GET
P_PressureChA := THIS^.rCurrentPressureInBarA;
END_GET
END_PROPERTY

{warning 'Eigenschaftenimplementierung hinzufügen'}
PROPERTY P_PressureChB : REAL
GET
P_PressureChB := THIS^.rCurrentPressureInBarB;
END_GET
END_PROPERTY

{warning 'Eigenschaftenimplementierung hinzufügen'}
PROPERTY P_PressureOk : BOOL
GET
//P_PRessureOk := ABS(rSetPressure - P_WorkPressure) < rEndPosTol;
END_GET
END_PROPERTY

{warning 'Eigenschaftenimplementierung hinzufügen'}
PROPERTY P_ReadyState : BOOL
GET
P_ReadyState := THIS^.stSeqCtrlGeneral.eActiveSeqState = E_SEQ_GENERAL.READY;
END_GET
END_PROPERTY

PROPERTY P_SpeedInMmPerSecond : REAL
GET
P_SpeedInMmPerSecond := THIS^.rCurrentSpeedInMmPerS;
END_GET
END_PROPERTY

{warning 'Eigenschaftenimplementierung hinzufügen'}
PROPERTY P_SpeedInPercent : LREAL
GET
P_SpeedInPercent := THIS^.rSpeedInPercentToSet;
END_GET
END_PROPERTY

PROPERTY P_StrokeLength : REAL
GET
P_StrokeLength := THIS^.rStrokeLength;
END_GET
END_PROPERTY

{warning 'Eigenschaftenimplementierung hinzufügen'}
PROPERTY P_StrokeLengthInitialized : BOOL
GET
P_StrokeLengthInitialized := THIS^.bStrokeLengthInitialized;
END_GET
SET
THIS^.bStrokeLengthInitialized := P_StrokeLengthInitialized;
END_SET
END_PROPERTY

PROPERTY P_WorkPressure : REAL
GET
P_WorkPressure := THIS^.rCurrentPressureInBar;
END_GET
END_PROPERTY

END_FUNCTION_BLOCK

// ---- POUs/MAIN.TcPOU
PROGRAM MAIN
VAR   
 	
END_VAR

END_PROGRAM

// ---- SUBSTATION/STATION_NEST/POU/FB_SEQ_PROCESS_NEST1.TcPOU
FUNCTION_BLOCK FB_SEQ_PROCESS_NEST1 IMPLEMENTS I_PROCESS_NEST1
VAR_INPUT
  bDoubleActing:                                          BOOL;
  rSpeedEfficiencyFactor:                                 REAL;
  uiRecordDelay:                                          UINT;
END_VAR
VAR_OUTPUT
  rMaxSpeedInMmPerSHP:                                    REAL := 999;
  rMaxSpeedInMmPerSWP:                                    REAL := 999;
END_VAR
VAR //General
	{attribute 'instance-path'} 
  {attribute 'noinit'} 
	strInstancePath:									                      STRING;
	bInit: 												                          BOOL:=TRUE;
	strFullObjectPath: 								                      STRING;
	stEvent:											                          ST_EVENT;
	bAck:												                            BOOL;
	bEnable:                                                BOOL;
END_VAR
VAR   // From FB_init	
	itfOpMode:											                        I_OP_MODE; 
  itfEventLogger:                                         I_EVENT_LOGGER; 
  itfTimer:                                               I_CLOCK;
  itfCounterCyl:                                          I_CYLINDER_DA_COUNTER;
  itfTestCyl:                                             I_CYLINDER_DA_TESTDEV1;
  itfCounterCylPump:                                      I_PUMP_WITH_BYPASS;
  itfTestCylPump:                                         I_PUMP;
  itfPump2Pressure:                                       I_PRV_PROP;
  itfPump3Pressure:                                       I_PRV_PROP;
  itfPump4Pressure:                                       I_PRV_PROP;
END_VAR                                      				
VAR	// Step chain control                				
  eSeq, eLastSeq, eNextSeq:					                      E_SEQ_PROCESS; 
  uiSnippetSeq, uiLastSnippetSeq:                         UINT := 0;
                  				
  //eActiveSeqState, eLastActiveSeqState:                 E_SEQ_GENERAL;
	(*
  iInternalSeqStateCase, iLastInternalSeqStateCase:       INT:=0;       
	tonDelay, tonTimeOut, tonStepTime:						          TON;
	tDelay:													                        TIME := T#100MS;
	tTimeOut:												                        TIME := T#100MS;
	tTimeOutExt:											                      TIME := T#100MS;
	bDelayActive, bTimeOutActiveQuit, bTimeOutActiveNoQuit:	BOOL;//Timer Option
	bActiveStep, bDebugAcitve, bDebugNext:					        BOOL;//Debug Option
	i:														                          INT;
 	iError:													                        INT; //ERROR-CODE                    	                   		
	listLastSteps:											                    ARRAY[0..49] OF ST_LAST_STEPS;	
	strExtraInfo:											                      STRING; 
	eStep_Type:												                      E_STEP_STATE_TYPE; 
	bDebugModeActive:										                    BOOL;   
	bWaitForBreakpoint:										                  BOOL;
	bBreakpointActive:										                  BOOL;
	bDebugResume:											                      BOOL;   
	listBreakpoint:											                    ARRAY[0..10] OF  INT;    
*)
i:														                            INT;
ii:                                                       INT;
stSeqCtrlGeneral:											                    ST_SEQ_CTRL_GEN;     	
END_VAR                                             		
VAR                                                 		
	bMethodeFromExtStarted:									                BOOL;
	bMethodeFromExtActive:									                BOOL;
	bMethodeFromExtDone:									                  BOOL;
	strTemp:												                        STRING;
END_VAR   
VAR
  strSerialNr:                                            STRING;
  udiCurrentCycle:                                        UDINT := 1;
  lrLastPos:                                              LREAL;
  rTargetLowPressureInBar:                                REAL;
  // Max Speed determination
  lrTotalSpeed:                                           LREAL := 0.0;
  udiSpeedDividend:                                       UDINT := 0;
  listSpeed:                                              ARRAY [1..6] OF REAL;
END_VAR    
VAR // Input variables
  bCylinderDecoupled:                                     BOOL := TRUE;
  uiVentCount:                                            UINT;
  udiERCycles:                                            UDINT;
  udiERTotalCycles:                                       UDINT := 0;
  stERParams:                                             ST_RECIPE_ENDURANCE_RUN;
  stBPDParams:                                            ST_RECIPE_BREAK_PRESSURE;
  stLT1Params:                                            ST_RECIPE_LEAK_TEST1;
  stLT2Params:                                            ST_RECIPE_LEAK_TEST2;
  uiCurrentNokLimitInPercent:                             UINT;
  rCurrentNokDifference:                                  REAL;
  lrStartPos:                                             LREAL;
  siLT2TestDirection:                                     SINT;
  lrStartReservoirPressure:                               LREAL;
  lrStartPressureA:                                       LREAL;
  lrStartPressureB:                                       LREAL;
  sTimer:                                                 STRING;
  rWorkForceATmp:                                         REAL;
  rWorkForceBTmp:                                         REAL;
  rLoadForceATmp:                                         REAL;
  rLoadForceBTmp:                                         REAL;
END_VAR      
VAR
  lrDistanceInM:                                          LREAL := 0.0;
  lrLastRecordPos:                                        LREAL := 0.0;
  uiRecordDelayCycleCount:                                UINT := 0;
END_VAR    	
VAR_TEMP                    	
	iTemp:											                            INT;
END_VAR

// Set FBs and Interfaces ready after switch internal step
IF stSeqCtrlGeneral.iInternalSeqStateCase <> stSeqCtrlGeneral.iLastInternalSeqStateCase AND NOT stSeqCtrlGeneral.bExitSetReadyState THEN
  uiSnippetSeq := 0;
  stSeqCtrlGeneral.bExitSetReadyState := TRUE
                                         AND itfCounterCyl.M_SetReady()
                                         AND itfTestCyl.M_SetReady()
                                         AND itfCounterCylPump.M_SetReady()
                                         AND itfTestCylPump.M_SetReady()
                                         AND uiSnippetSeq = 0;
  IF TRUE
  AND (stERParams.rSpeedA > THIS^.rMaxSpeedInMmPerSWP * THIS^.rSpeedEfficiencyFactor
  OR stERParams.rSpeedB > THIS^.rMaxSpeedInMmPerSHP * THIS^.rSpeedEfficiencyFactor)
  THEN
    stSeqCtrlGeneral.bExitSetReadyState := TRUE
                                           AND itfPump2Pressure.M_SetReady()
                                           AND itfPump3Pressure.M_SetReady()
                                           AND itfPump4Pressure.M_SetReady();
  END_IF
  IF NOT stSeqCtrlGeneral.bExitSetReadyState THEN 
    RETURN; 
  END_IF
END_IF

stSeqCtrlGeneral.strObject := F_CreateObjectName(strInstancePath);
sTimer := itfTimer.M_GetTimerET(bCustomFormat:= FALSE, sFormat:= '');

// First method call
_m_SequenceManager();
//_m_SaveLastStep();

CASE eSeq OF 
  E_SEQ_VALVE.BASE:;
  
	E_SEQ_PROCESS.INIT: _m_Seq_INIT();
		IF TRUE
		AND (stSeqCtrlGeneral.eActiveSeqState = E_SEQ_GENERAL.DONE) 
		THEN
			eSeq := E_SEQ_PROCESS.BASE;
		END_IF
		
	E_SEQ_PROCESS.SETUP:;
  
	// Process
	E_SEQ_PROCESS.MEASURE_STROKE_LENGTH: _m_Seq_MEASURE_STROKE_LENGTH();
    IF TRUE
		AND (stSeqCtrlGeneral.eActiveSeqState = E_SEQ_GENERAL.DONE) 
		THEN
			eSeq := E_SEQ_PROCESS.BASE;
		END_IF
  
  E_SEQ_PROCESS.VENT_CYLINDER: _m_Seq_VENT_CYLINDER();
    IF TRUE
		AND (stSeqCtrlGeneral.eActiveSeqState = E_SEQ_GENERAL.DONE) 
		THEN
			eSeq := E_SEQ_PROCESS.BASE;
		END_IF
  
  E_SEQ_PROCESS.MOVE_TO_SET_POS: _m_Seq_MOVE_TO_SET_POS();
    IF TRUE
		AND (stSeqCtrlGeneral.eActiveSeqState = E_SEQ_GENERAL.DONE) 
		THEN
			eSeq := E_SEQ_PROCESS.BASE;
		END_IF
  
  E_SEQ_PROCESS.BREAK_PRESSURE_DET: _m_Seq_BREAK_PRESSURE_DET();
    IF TRUE
		AND (stSeqCtrlGeneral.eActiveSeqState = E_SEQ_GENERAL.DONE) 
		THEN
			eSeq := E_SEQ_PROCESS.BASE;
		END_IF
  
  E_SEQ_PROCESS.LEAK_TEST_1: _m_Seq_LEAK_TEST_1();
    IF TRUE
		AND (stSeqCtrlGeneral.eActiveSeqState = E_SEQ_GENERAL.DONE) 
		THEN
			eSeq := E_SEQ_PROCESS.BASE;
		END_IF
  
  E_SEQ_PROCESS.LEAK_TEST_2: _m_Seq_LEAK_TEST_2();
    IF TRUE
		AND (stSeqCtrlGeneral.eActiveSeqState = E_SEQ_GENERAL.DONE) 
		THEN
			eSeq := E_SEQ_PROCESS.BASE;
		END_IF
  
  E_SEQ_PROCESS.ENDURANCE_RUN: _m_Seq_ENDURANCE_RUN();
    IF TRUE
		AND (stSeqCtrlGeneral.eActiveSeqState = E_SEQ_GENERAL.DONE) 
		THEN
			eSeq := E_SEQ_PROCESS.BASE;
		END_IF
    
  E_SEQ_PROCESS.MAX_SPEED_RECORD: _m_Seq_MAX_SPEED_RECORD();
    IF TRUE
		AND (stSeqCtrlGeneral.eActiveSeqState = E_SEQ_GENERAL.DONE) 
		THEN
      eSeq := eNextSeq := E_SEQ_PROCESS.BASE;
		END_IF

  E_SEQ_PROCESS.STOP_ENGINE: _m_Seq_STOP_ENGINE();
    IF TRUE
		AND (stSeqCtrlGeneral.eActiveSeqState = E_SEQ_GENERAL.DONE) 
		THEN
			eSeq := E_SEQ_PROCESS.BASE;
		END_IF
    
  E_SEQ_PROCESS.STOP: _m_Seq_STOP();
    IF TRUE
		AND (stSeqCtrlGeneral.eActiveSeqState = E_SEQ_GENERAL.DONE) 
		THEN
			eSeq := E_SEQ_PROCESS.BASE;
		END_IF
    
  E_SEQ_PROCESS.RESET_DISTANCE: _m_Seq_RESET_DISTANCE();
    IF TRUE
		AND stSeqCtrlGeneral.eActiveSeqState = E_SEQ_GENERAL.DONE
		THEN
			eSeq := E_SEQ_PROCESS.BASE;
		END_IF
    
  E_SEQ_PROCESS.MOVE_CYL_TO_HP: _m_Seq_MOVE_CYL1_TO_HP();
    IF TRUE
		AND stSeqCtrlGeneral.eActiveSeqState = E_SEQ_GENERAL.DONE
		THEN
			eSeq := E_SEQ_PROCESS.BASE;
		END_IF
    
  // End
	E_SEQ_PROCESS.END:;
	E_SEQ_PROCESS.ERROR_SEQ:;	
END_CASE

strTemp:=TO_STRING(eSeq);

METHOD PRIVATE _m_DebugManager
VAR_INPUT
	iStepID: int;
END_VAR
IF TRUE
AND THIS^.stSeqCtrlGeneral.bDebugModeActive 
AND NOT THIS^.stSeqCtrlGeneral.bActiveStep
THEN


THIS^.stSeqCtrlGeneral.bBreakpointActive:=FALSE;

FOR i:=0 TO 10 DO
	
	IF TRUE
	AND iStepID=THIS^.stSeqCtrlGeneral.listBreakpoint[i] 
	AND iStepID<>0
	THEN
		EXIT;
	END_IF
END_FOR
IF (i<=10) THEN
	THIS^.stSeqCtrlGeneral.bBreakpointActive:=TRUE;
END_IF

END_IF
END_METHOD

METHOD PRIVATE _m_Delay : BOOL
VAR_INPUT
	DelayTime:	TIME;
END_VAR
THIS^.stSeqCtrlGeneral.bDelayActive := TRUE;
THIS^.stSeqCtrlGeneral.tDelay := DelayTime;

_m_Delay := THIS^.stSeqCtrlGeneral.tonDelay.Q;
END_METHOD

METHOD PRIVATE _m_DistanceRecord : BOOL
VAR_INPUT
END_VAR
// The last position was set at the first call
IF THIS^.uiRecordDelayCycleCount = 0 THEN
  THIS^.lrLastRecordPos := THIS^.itfTestCyl.P_Position;
END_IF

IF THIS^.uiRecordDelayCycleCount >= 100 THEN
THIS^.lrDistanceInM := THIS^.lrDistanceInM + (ABS(THIS^.itfTestCyl.P_Position - THIS^.lrLastRecordPos) / 1000);

THIS^.lrLastRecordPos := THIS^.itfTestCyl.P_Position;
THIS^.uiRecordDelayCycleCount := 1;
END_IF


THIS^.uiRecordDelayCycleCount := THIS^.uiRecordDelayCycleCount + 1;
END_METHOD

METHOD PRIVATE _m_GeneralStepSetting : BOOL
VAR_INPUT
	StepType:			    	E_STEP_STATE_TYPE;
	InfoTextID:					STRING(20);
	EnableDebug:	   			BOOL;	
	
END_VAR
IF THIS^.stSeqCtrlGeneral.bActiveStep THEN
	THIS^.stSeqCtrlGeneral.eStep_Type:=StepType;
	THIS^.stSeqCtrlGeneral.strExtraInfo:= GenLib.F_RET_TXTLIST_ENTRY(strPortNr:='851',strID:='',strTxtLstName:=InfoTextID);
END_IF
END_METHOD

METHOD PRIVATE _m_LeakTest1_LeakDet : BOOL
VAR_INPUT
END_VAR
_m_LeakTest1_LeakDet := THIS^.uiSnippetSeq = 999;

IF TRUE 
AND THIS^.uiSnippetSeq <> THIS^.uiLastSnippetSeq 
THEN
  IF NOT _m_ResetDelayTimer() THEN
    RETURN;
	END_IF
END_IF

THIS^.uiLastSnippetSeq := THIS^.uiSnippetSeq;

CASE THIS^.uiSnippetSeq OF
  0:
    IF TRUE
    AND _m_ResetDelayTimer()
		THEN 
      THIS^.uiSnippetSeq := 10;
		END_IF
  
  10:
    IF TRUE
    AND _m_Delay(DelayTime:= UINT_TO_TIME(THIS^.uiRecordDelay * 1000))
		THEN 
      THIS^.lrStartPos := THIS^.itfTestCyl.P_Position;
      THIS^.uiSnippetSeq := 20;
		END_IF
    
  20:
    IF TRUE
    AND _m_Delay(DelayTime:= UDINT_TO_TIME(THIS^.stLT1Params.udiDurationPerTest * 60000))
		THEN 
      THIS^.uiSnippetSeq := 999;
		END_IF
    IF ABS(THIS^.lrStartPos - THIS^.itfTestCyl.P_Position) > ABS(THIS^.stLT1Params.rNokLimit) THEN
      THIS^.itfEventLogger.M_ErrorMsg(udiID:= 10170, sMsg:= 'NOK-Limit wurde überschritten!', bWithConfirmation:= FALSE);
      THIS^.stSeqCtrlGeneral.eActiveSeqState := E_SEQ_GENERAL.ERROR; // Error step
		END_IF
    THIS^.rCurrentNokDifference := ABS(THIS^.lrStartPos - THIS^.itfTestCyl.P_Position);
    THIS^.uiCurrentNokLimitInPercent := TO_UINT(100 / ABS(THIS^.stLT1Params.rNokLimit) * THIS^.rCurrentNokDifference);
END_CASE
END_METHOD

METHOD PRIVATE _m_LeakTest2_LeakDet : BOOL
VAR_INPUT
END_VAR
VAR
  rV0:                  REAL := 75;
  rTmpVal:              REAL;
END_VAR

// Formula for Leak Test 2
// V0 Speicher = 75 cm³ (ml)
// P0 Speicher = 95 bar
// P2 (Anfangsdruck) = 354.4 bar
// P1 (Enddruck) = 353.7 bar
// Ergebnis = 0.01 cm³ (ml)

// DeltaV = V0 * SQRT((P0 / P2) * ((P2 / P1) - 1))
_m_LeakTest2_LeakDet := THIS^.uiSnippetSeq = 999;

IF TRUE 
AND THIS^.uiSnippetSeq <> THIS^.uiLastSnippetSeq 
THEN
  IF NOT _m_ResetDelayTimer() THEN
    RETURN;
	END_IF
END_IF

THIS^.uiLastSnippetSeq := THIS^.uiSnippetSeq;

CASE THIS^.uiSnippetSeq OF
  0:
    IF TRUE
    AND _m_ResetDelayTimer()
		THEN 
      THIS^.uiSnippetSeq := 10;
		END_IF
  
  10:
    IF TRUE
    AND _m_Delay(DelayTime:= UINT_TO_TIME(THIS^.uiRecordDelay * 1000))
		THEN 
      THIS^.lrStartPressureA := THIS^.itfTestCyl.P_PressureChA;
      THIS^.lrStartPressureB := THIS^.itfTestCyl.P_PressureChB;
      THIS^.lrStartReservoirPressure := THIS^.itfTestCyl.P_ReservoirPressure;
      THIS^.uiSnippetSeq := 20;
		END_IF
    
  20:
    IF TRUE
		THEN 
      IF TRUE
         AND ((THIS^.siLT2TestDirection = 1 AND THIS^.lrStartPressureA <= 10) 
         OR (THIS^.siLT2TestDirection = -1 AND THIS^.lrStartPressureB <= 10)
         OR THIS^.lrStartReservoirPressure < 10
         OR (THIS^.siLT2TestDirection <> -1 AND THIS^.siLT2TestDirection <> 1))
      THEN
        THIS^.stSeqCtrlGeneral.eActiveSeqState := E_SEQ_GENERAL.ERROR;
      ELSE
        THIS^.uiSnippetSeq := 30;
      END_IF
		END_IF
    
  30: // Direction choice
    IF siLT2TestDirection = -1 THEN
      THIS^.uiSnippetSeq := 40;
    ELSIF siLT2TestDirection = 1 THEN
      THIS^.uiSnippetSeq := 50;
    ELSE
      THIS^.stSeqCtrlGeneral.eActiveSeqState := E_SEQ_GENERAL.ERROR;
		END_IF
    
  40:
    IF TRUE
    AND _m_Delay(DelayTime:= UDINT_TO_TIME(THIS^.stLT2Params.udiDurationPerTest * 60000))
		THEN 
      THIS^.uiSnippetSeq := 999;
		END_IF
    IF ABS(THIS^.rCurrentNokDifference) > ABS(THIS^.stLT2Params.rNokLimit) THEN
      THIS^.itfEventLogger.M_ErrorMsg(udiID:= 10170, sMsg:= 'NOK-Limit wurde überschritten!', bWithConfirmation:= FALSE);
      THIS^.stSeqCtrlGeneral.eActiveSeqState := E_SEQ_GENERAL.ERROR; // Error step
		END_IF
    rTmpVal := F_RoundREAL(rValue:= (THIS^.lrStartReservoirPressure / THIS^.lrStartPressureB) * ((THIS^.lrStartPressureB / THIS^.itfTestCyl.P_PressureChB) - 1), 
                           uiDezimalPlace:= 6);
    IF ABS(rTmpVal) <> 0.0 THEN
      THIS^.rCurrentNokDifference := 75 * SQRT(ABS(rTmpVal));
    ELSE
      THIS^.rCurrentNokDifference := 0;
    END_IF
    THIS^.uiCurrentNokLimitInPercent := TO_UINT(100 / ABS(THIS^.stLT2Params.rNokLimit) * THIS^.rCurrentNokDifference);
    
  50:
    IF TRUE
    AND _m_Delay(DelayTime:= UDINT_TO_TIME(THIS^.stLT2Params.udiDurationPerTest * 60000))
		THEN 
      THIS^.uiSnippetSeq := 999;
		END_IF
    IF ABS(THIS^.rCurrentNokDifference) > ABS(THIS^.stLT2Params.rNokLimit) THEN
      THIS^.itfEventLogger.M_ErrorMsg(udiID:= 10170, sMsg:= 'NOK-Limit wurde überschritten!', bWithConfirmation:= FALSE);
      THIS^.stSeqCtrlGeneral.eActiveSeqState := E_SEQ_GENERAL.ERROR; // Error step
		END_IF
    rTmpVal := F_RoundREAL(rValue:= (THIS^.lrStartReservoirPressure / THIS^.lrStartPressureA) * ((THIS^.lrStartPressureA / THIS^.itfTestCyl.P_PressureChA) - 1), 
                           uiDezimalPlace:= 6);
    IF ABS(rTmpVal) <> 0.0 THEN
      THIS^.rCurrentNokDifference := 75 * SQRT(ABS(rTmpVal));
    ELSE
      THIS^.rCurrentNokDifference := 0;
    END_IF
    THIS^.uiCurrentNokLimitInPercent := TO_UINT(100 / ABS(THIS^.stLT2Params.rNokLimit) * THIS^.rCurrentNokDifference);
END_CASE
END_METHOD

METHOD PRIVATE _m_ResetDelayTimer : BOOL
_m_ResetDelayTimer := THIS^.stSeqCtrlGeneral.tonDelay.ET = T#0MS;

THIS^.stSeqCtrlGeneral.tonDelay(IN:= FALSE);
END_METHOD

METHOD PRIVATE _m_SaveLastStep : BOOL
VAR_INPUT
END_VAR
VAR
	i: dint;
END_VAR
IF NOT THIS^.stSeqCtrlGeneral.bActiveStep THEN
	
	FOR i:=49 TO 1 BY -1 DO
			stSeqCtrlGeneral.listLastSteps[i].strStepName:=stSeqCtrlGeneral.listLastSteps[i-1].strStepName;
			stSeqCtrlGeneral.listLastSteps[i].tStepTime:=stSeqCtrlGeneral.listLastSteps[i-1].tStepTime;
			stSeqCtrlGeneral.listLastSteps[i].tDelayTime:=stSeqCtrlGeneral.listLastSteps[i-1].tDelayTime;
	END_FOR
	stSeqCtrlGeneral.listLastSteps[0].strStepName:=TO_STRING(THIS^.eSeq);
	stSeqCtrlGeneral.listLastSteps[1].tStepTime:=THIS^.stSeqCtrlGeneral.tonStepTime.ET;
	stSeqCtrlGeneral.listLastSteps[1].tStepTime:=THIS^.stSeqCtrlGeneral.tonDelay.ET;
ELSE
	stSeqCtrlGeneral.listLastSteps[0].tStepTime:=THIS^.stSeqCtrlGeneral.tonStepTime.ET;
	stSeqCtrlGeneral.listLastSteps[0].tDelayTime:=THIS^.stSeqCtrlGeneral.tonDelay.ET;	
END_IF
END_METHOD

METHOD PRIVATE _m_Seq_BREAK_PRESSURE_DET : E_SEQ_PROCESS
VAR_INPUT
END_VAR
VAR
  ActiveSeq:    STRING;
END_VAR
//THIS^._m_GeneralStepSetting(StepType:=E_STEP_STATE_TYPE.INIT,
ActiveSeq := TO_STRING(THIS^.eSeq);

CASE THIS^.stSeqCtrlGeneral.eActiveSeqState OF
E_SEQ_GENERAL.READY:;

	
E_SEQ_GENERAL.EXECUTE:;
	IF TRUE
	AND _m_Delay(T#1S)
	THEN
		THIS^.stSeqCtrlGeneral.eActiveSeqState := E_SEQ_GENERAL.RESET;
	END_IF
  
E_SEQ_GENERAL.RESET:;
	stSeqCtrlGeneral.iInternalSeqStateCase := 0;
	IF TRUE
	THEN
		THIS^.stSeqCtrlGeneral.eActiveSeqState := E_SEQ_GENERAL.BUSY;
	END_IF
  
E_SEQ_GENERAL.BUSY:;
	CASE THIS^.stSeqCtrlGeneral.iInternalSeqStateCase OF
    0: // Check if enable
      IF TRUE
      AND THIS^.bEnable 
      THEN
        THIS^.stSeqCtrlGeneral.iInternalSeqStateCase := 10; 
      ELSE
        THIS^.stSeqCtrlGeneral.iInternalSeqStateCase := 9999; 
			END_IF

    10: // Disable low pressure mode
      IF TRUE 
			AND THIS^.itfTestCyl.M_LowPressureMode(bSet:= FALSE, ePressureType:= E_PRESSURE_TYPE.VALUE, rWorkPressure:= 0)
			THEN 
				THIS^.stSeqCtrlGeneral.iInternalSeqStateCase := 20; 
			END_IF
      
    20: // Disable pump 2
      IF TRUE 
			AND THIS^.itfTestCyl.M_Pump2Add(bAdd:= FALSE)
      AND THIS^.itfPump2Pressure.M_SetLimit(ePressureType:= E_PRESSURE_TYPE.PERCENT, rLimit:= 0)
			THEN
        THIS^.stSeqCtrlGeneral.iInternalSeqStateCase := 30; 
			END_IF
      
    30: // Disable pump 3
      IF TRUE 
			AND THIS^.itfTestCyl.M_Pump3Add(bAdd:= FALSE)
      AND THIS^.itfPump3Pressure.M_SetLimit(ePressureType:= E_PRESSURE_TYPE.PERCENT, rLimit:= 0)
			THEN
        THIS^.stSeqCtrlGeneral.iInternalSeqStateCase := 40; 
			END_IF
      
    40: // Disable pump 4
      IF TRUE 
			AND THIS^.itfTestCyl.M_Pump4Add(bAdd:= FALSE)
      AND THIS^.itfPump4Pressure.M_SetLimit(ePressureType:= E_PRESSURE_TYPE.PERCENT, rLimit:= 0)
			THEN
        IF THIS^.bDoubleActing THEN
          THIS^.stSeqCtrlGeneral.iInternalSeqStateCase := 50; 
        ELSE
          THIS^.stSeqCtrlGeneral.iInternalSeqStateCase := 60; 
        END_IF
			END_IF
      
    50:	// Move test cylinder to HP
      IF TRUE  
      AND _m_Delay(DelayTime:= T#3S)
      AND THIS^.itfTestCyl.M_ToHP(ePressureType:= E_PRESSURE_TYPE.FORCE, 
                                  rWorkPressure:= 2 * 1000, 
                                  bPressureRegulation:= FALSE,
                                  eSpeedType:= E_SPEED_TYPE.PERCENT, 
                                  rSpeed:= 50)
      AND THIS^.itfTestCyl.P_Position <= THIS^.stBPDParams.rEndPosTol
      AND THIS^.itfTestCyl.P_SpeedInMmPerSecond < 0.1
			THEN 
        THIS^.stSeqCtrlGeneral.iInternalSeqStateCase := 60;
			END_IF
      
    60:	// Stop
      IF TRUE  
      AND THIS^.itfTestCyl.M_Stop()
			THEN 
        THIS^.stSeqCtrlGeneral.iInternalSeqStateCase := 70;
			END_IF
      
    70:	// Set work pressure zero
      IF TRUE  
      AND THIS^.itfTestCyl.M_SetWorkPressureZero()
			THEN 
        THIS^.stSeqCtrlGeneral.iInternalSeqStateCase := 80;
			END_IF
      
		80:	// Open low pressure valve, set limit zero and move counter cylinder to HP
      IF TRUE 
      AND _m_Delay(DelayTime:= T#25S)
      AND THIS^.itfCounterCyl.M_ToHP(ePressureType:= E_PRESSURE_TYPE.BAR, 
                                     rWorkPressure:= 10, 
                                     bPressureRegulation:= FALSE,
                                     eSpeedType:= E_SPEED_TYPE.PERCENT, 
                                     rSpeed:= 50)
      AND THIS^.itfTestCyl.M_LowPressureMode(bSet:= TRUE, ePressureType:= E_PRESSURE_TYPE.BAR, rWorkPressure:= 0)
			THEN 
        THIS^.rTargetLowPressureInBar := THIS^.stBPDParams.rIncreaseValueInBar;
        THIS^.stSeqCtrlGeneral.iInternalSeqStateCase := 90;
			END_IF
      
    90:	// Stop counter cylinder
      IF TRUE 
      AND _m_Delay(T#1S)
      AND THIS^.itfCounterCyl.M_Stop()
			THEN 
        THIS^.stSeqCtrlGeneral.iInternalSeqStateCase := 100;
			END_IF
  
		100:	// Move test cylinder to WP
      IF TRUE 
      AND THIS^.itfTestCyl.M_ToWP(ePressureType:= E_PRESSURE_TYPE.BAR, 
                                  rWorkPressure:= 100, 
                                  bPressureRegulation:= FALSE,
                                  eSpeedType:= E_SPEED_TYPE.PERCENT, 
                                  rSpeed:= 100)
			THEN 
				THIS^.stSeqCtrlGeneral.iInternalSeqStateCase := 110; 
			END_IF
      
    110:	// Set pressure
      IF TRUE 
			AND THIS^.itfTestCyl.M_LowPressureMode(bSet:= TRUE, ePressureType:= E_PRESSURE_TYPE.BAR, rWorkPressure:= THIS^.rTargetLowPressureInBar)
			THEN 
				THIS^.stSeqCtrlGeneral.iInternalSeqStateCase := 120; 
			END_IF
      
    120:	// Increase time
      IF TRUE 
			AND _m_Delay(DelayTime:= REAL_TO_TIME(THIS^.stBPDParams.rIncreaseInterval * 1000))
			THEN 
				THIS^.stSeqCtrlGeneral.iInternalSeqStateCase := 121; 
			END_IF
      
    121:	// Check if cylinder moving or in end position
      IF TRUE 
			AND ABS(THIS^.itfTestCyl.P_SpeedInMmPerSecond) < ABS(THIS^.stBPDParams.rMinSpeedInMmPerS)
      AND THIS^.itfTestCyl.P_Position < THIS^.itfTestCyl.P_StrokeLength - ABS(THIS^.stBPDParams.rEndPosTol)
			THEN 
        THIS^.rTargetLowPressureInBar := THIS^.rTargetLowPressureInBar + ABS(THIS^.stBPDParams.rIncreaseValueInBar);
				THIS^.stSeqCtrlGeneral.iInternalSeqStateCase := 110; 
      ELSIF TRUE 
			AND ABS(THIS^.itfTestCyl.P_SpeedInMmPerSecond) < ABS(THIS^.stBPDParams.rMinSpeedInMmPerS)
      AND THIS^.itfTestCyl.P_Position >= THIS^.itfTestCyl.P_StrokeLength - ABS(THIS^.stBPDParams.rEndPosTol)
      THEN
        THIS^.stSeqCtrlGeneral.iInternalSeqStateCase := 130; 
      ELSE
        THIS^.stSeqCtrlGeneral.iInternalSeqStateCase := 120; 
			END_IF
      
    130:  // Check if test reverse break pressure or exit sequence
      IF TRUE
      AND THIS^.bDoubleActing 
      AND THIS^.itfTestCyl.P_Position > THIS^.itfTestCyl.P_StrokeLength - ABS(THIS^.stBPDParams.rEndPosTol + 5) 
      THEN
        THIS^.stSeqCtrlGeneral.iInternalSeqStateCase := 200; 
      ELSE
        THIS^.stSeqCtrlGeneral.iInternalSeqStateCase := 1000; 
			END_IF
      
    (*Testing double acting cylinder to HP*)
    200:	// Stop
      IF TRUE  
      AND THIS^.itfTestCyl.M_Stop()
			THEN 
        THIS^.stSeqCtrlGeneral.iInternalSeqStateCase := 210;
			END_IF
      
		210:	// Set limit zero
      IF TRUE 
      AND _m_Delay(DelayTime:= T#3S)
      AND THIS^.itfTestCyl.M_LowPressureMode(bSet:= TRUE, ePressureType:= E_PRESSURE_TYPE.BAR, rWorkPressure:= 0)
			THEN 
        THIS^.rTargetLowPressureInBar := THIS^.stBPDParams.rIncreaseValueInBar;
        THIS^.stSeqCtrlGeneral.iInternalSeqStateCase := 220;
			END_IF
  
		220:	// Move test cylinder to HP
      IF TRUE 
      AND THIS^.itfTestCyl.M_ToHP(ePressureType:= E_PRESSURE_TYPE.BAR, 
                                  rWorkPressure:= 100, 
                                  bPressureRegulation:= FALSE,
                                  eSpeedType:= E_SPEED_TYPE.PERCENT, 
                                  rSpeed:= 100)
			THEN 
				THIS^.stSeqCtrlGeneral.iInternalSeqStateCase := 230; 
			END_IF
      
    230:	// Set pressure
      IF TRUE 
			AND THIS^.itfTestCyl.M_LowPressureMode(bSet:= TRUE, ePressureType:= E_PRESSURE_TYPE.BAR, rWorkPressure:= THIS^.rTargetLowPressureInBar)
			THEN 
				THIS^.stSeqCtrlGeneral.iInternalSeqStateCase := 240; 
			END_IF
      
    240:	// Increase time
      IF TRUE 
			AND _m_Delay(DelayTime:= REAL_TO_TIME(THIS^.stBPDParams.rIncreaseInterval * 1000))
			THEN 
				THIS^.stSeqCtrlGeneral.iInternalSeqStateCase := 241; 
			END_IF
      
    241:	// Check if cylinder moving or in end position
      IF TRUE 
			AND ABS(THIS^.itfTestCyl.P_SpeedInMmPerSecond) < ABS(THIS^.stBPDParams.rMinSpeedInMmPerS)
      AND THIS^.itfTestCyl.P_Position > ABS(THIS^.stBPDParams.rEndPosTol)
			THEN 
        THIS^.rTargetLowPressureInBar := THIS^.rTargetLowPressureInBar + ABS(THIS^.stBPDParams.rIncreaseValueInBar);
				THIS^.stSeqCtrlGeneral.iInternalSeqStateCase := 230; 
      ELSIF TRUE 
			AND ABS(THIS^.itfTestCyl.P_SpeedInMmPerSecond) < ABS(THIS^.stBPDParams.rMinSpeedInMmPerS)
      AND THIS^.itfTestCyl.P_Position <= ABS(THIS^.stBPDParams.rEndPosTol)
      THEN
        THIS^.stSeqCtrlGeneral.iInternalSeqStateCase := 1000; 
      ELSE
        THIS^.stSeqCtrlGeneral.iInternalSeqStateCase := 240; 
			END_IF
      
    1000: // Exit seq - Stop
      IF TRUE
      AND _m_Delay(DelayTime:= T#1S) 
      AND THIS^.itfTestCyl.M_Stop()
      AND THIS^.itfCounterCyl.M_Stop()
			THEN 
				THIS^.stSeqCtrlGeneral.iInternalSeqStateCase := 1010;
			END_IF
      
    1010: // Set pressure
      IF TRUE 
			AND THIS^.itfCounterCyl.M_SetWorkPressureZero()
      AND THIS^.itfTestCyl.M_SetWorkPressureZero()
			THEN 
				THIS^.stSeqCtrlGeneral.iInternalSeqStateCase := 9999; 
			END_IF
      
	ELSE
		THIS^.stSeqCtrlGeneral.eActiveSeqState := E_SEQ_GENERAL.DONE;  
	END_CASE
	THIS^.stSeqCtrlGeneral.strExtraInfo := CONCAT('Internal state: ', TO_STRING(THIS^.stSeqCtrlGeneral.iInternalSeqStateCase));
E_SEQ_GENERAL.DONE:;
E_SEQ_GENERAL.ERROR:;
E_SEQ_GENERAL.TIME_OUT:; 

IF TRUE
AND THIS^.stSeqCtrlGeneral.bTimeOutActiveQuit 
THEN
  THIS^.stSeqCtrlGeneral.strExtraInfo := 'Bitte quittieren und erneut testen';
  IF TRUE
  //AND itfOpMode.P_QUIT
  THEN
    THIS^.stSeqCtrlGeneral.eActiveSeqState := E_SEQ_GENERAL.EXECUTE;
	END_IF
  
END_IF

ELSE
  THIS^.stSeqCtrlGeneral.eActiveSeqState := E_SEQ_GENERAL.ERROR;
END_CASE
END_METHOD

METHOD PRIVATE _m_Seq_ENDURANCE_RUN : E_SEQ_PROCESS
VAR_INPUT
END_VAR
VAR
  ActiveSeq:            STRING;
END_VAR
//THIS^._m_GeneralStepSetting(StepType:=E_STEP_STATE_TYPE.INIT,
ActiveSeq := TO_STRING(THIS^.eSeq);

// Distance record
_m_DistanceRecord();

CASE THIS^.stSeqCtrlGeneral.eActiveSeqState OF
E_SEQ_GENERAL.READY:;

	
E_SEQ_GENERAL.EXECUTE:;
	IF TRUE
	AND _m_Delay(T#1S)
	THEN
		THIS^.stSeqCtrlGeneral.eActiveSeqState := E_SEQ_GENERAL.RESET;
	END_IF
  
E_SEQ_GENERAL.RESET:;
	stSeqCtrlGeneral.iInternalSeqStateCase := 0;
	IF TRUE
	THEN
    THIS^.udiCurrentCycle := 1;
		THIS^.stSeqCtrlGeneral.eActiveSeqState := E_SEQ_GENERAL.BUSY;
	END_IF
  
E_SEQ_GENERAL.BUSY:;
	CASE THIS^.stSeqCtrlGeneral.iInternalSeqStateCase OF
    0: // Check if enable
      IF TRUE
      AND THIS^.bEnable 
      THEN
        THIS^.stSeqCtrlGeneral.iInternalSeqStateCase := 10; 
      ELSE
        THIS^.stSeqCtrlGeneral.iInternalSeqStateCase := 9999; 
			END_IF
    
		10: // Disable low pressure mode
      IF TRUE 
			AND THIS^.itfTestCyl.M_LowPressureMode(bSet:= FALSE, ePressureType:= E_PRESSURE_TYPE.VALUE, rWorkPressure:= 0)
			THEN
        IF TRUE
        AND (THIS^.stERParams.rSpeedA > THIS^.rMaxSpeedInMmPerSWP * THIS^.rSpeedEfficiencyFactor
        OR (THIS^.bDoubleActing AND THIS^.stERParams.rSpeedB > THIS^.rMaxSpeedInMmPerSHP * THIS^.rSpeedEfficiencyFactor)) 
        THEN
          THIS^.stSeqCtrlGeneral.iInternalSeqStateCase := 11; 
        ELSE
          THIS^.stSeqCtrlGeneral.iInternalSeqStateCase := 15; 
				END_IF
			END_IF
      
    11: // Add pump 2
      IF TRUE 
			AND THIS^.itfTestCyl.M_Pump2Add(bAdd:= TRUE)
      AND THIS^.itfPump2Pressure.M_SetLimit(ePressureType:= E_PRESSURE_TYPE.PERCENT, rLimit:= 100)
			THEN
        THIS^.stSeqCtrlGeneral.iInternalSeqStateCase := 12; 
			END_IF
      
    12: // Add pump 3
      IF TRUE 
			AND THIS^.itfTestCyl.M_Pump3Add(bAdd:= TRUE)
      AND THIS^.itfPump3Pressure.M_SetLimit(ePressureType:= E_PRESSURE_TYPE.PERCENT, rLimit:= 100)
			THEN
        THIS^.stSeqCtrlGeneral.iInternalSeqStateCase := 13; 
			END_IF
      
    13: // Add pump 4
      IF TRUE 
			AND THIS^.itfTestCyl.M_Pump4Add(bAdd:= TRUE)
      AND THIS^.itfPump4Pressure.M_SetLimit(ePressureType:= E_PRESSURE_TYPE.PERCENT, rLimit:= 100)
			THEN
        THIS^.stSeqCtrlGeneral.iInternalSeqStateCase := 15; 
			END_IF

    15: // Choice step
      IF TRUE 
			THEN 
        IF TRUE
        AND THIS^.udiCurrentCycle > THIS^.udiERCycles 
        THEN
          THIS^.stSeqCtrlGeneral.iInternalSeqStateCase := 1000; 
        ELSE
          THIS^.stSeqCtrlGeneral.iInternalSeqStateCase := 20; 
				END_IF
			END_IF
      
    20: // Add low pressure circuit to counter cylinder
      IF TRUE 
			AND THIS^.itfCounterCyl.M_LowPressureCircuit(bAdd:= TRUE)
			THEN 
				THIS^.stSeqCtrlGeneral.iInternalSeqStateCase := 30; 
			END_IF
      
    30: // Stop
      IF TRUE
      AND _m_Delay(DelayTime:= REAL_TO_TIME(THIS^.stERParams.rDelay * 1000))
      AND THIS^.itfTestCyl.M_Stop()
      AND THIS^.itfCounterCyl.M_Stop()
			THEN 
        THIS^.stSeqCtrlGeneral.iInternalSeqStateCase := 40; 
			END_IF
      
    40: // Move to WP (Max position - 10)
      IF TRUE
      AND THIS^.itfTestCyl.M_ToWP(ePressureType:= E_PRESSURE_TYPE.FORCE, 
                                  rWorkPressure:= THIS^.stERParams.rWorkForceA * 1000, 
                                  bPressureRegulation:= TRUE,
                                  eSpeedType:= E_SPEED_TYPE.MM_PER_SECOND, 
                                  rSpeed:= THIS^.stERParams.rSpeedA)
      AND THIS^.itfCounterCyl.M_ToWP( ePressureType:= E_PRESSURE_TYPE.FORCE, 
                                      rWorkPressure:= THIS^.stERParams.rLoadForceA * 1000, 
                                      bPressureRegulation:= TRUE,
                                      eSpeedType:= E_SPEED_TYPE.PERCENT, 
                                      rSpeed:= 50)
			THEN 
        THIS^.stSeqCtrlGeneral.iInternalSeqStateCase := 50;
			END_IF
      
    50: // Move to WP (Max position - 10)
      IF TRUE
			THEN 
        IF THIS^.itfTestCyl.P_Position >= THIS^.itfTestCyl.P_StrokeLength - ABS(THIS^.stERParams.rTurningPointWP) THEN
				  THIS^.stSeqCtrlGeneral.iInternalSeqStateCase := 60; 
        END_IF
			END_IF
      
    60: // Stop
      IF TRUE
      AND _m_Delay(DelayTime:= REAL_TO_TIME(THIS^.stERParams.rDelay * 1000))
      AND THIS^.itfTestCyl.M_Stop()
      AND THIS^.itfCounterCyl.M_Stop()
			THEN 
        THIS^.stSeqCtrlGeneral.iInternalSeqStateCase := 70; 
			END_IF
      
    70: // Move to HP (Min position + 10)
      IF TRUE
			THEN 
        IF THIS^.bDoubleActing THEN
          THIS^.stSeqCtrlGeneral.iInternalSeqStateCase := 71;
        ELSE
          THIS^.stSeqCtrlGeneral.iInternalSeqStateCase := 72;
        END_IF
			END_IF
      
    71: // Move to HP (Min position + 10)
      IF TRUE
      AND THIS^.itfTestCyl.M_ToHP(ePressureType:= E_PRESSURE_TYPE.FORCE, 
                                  rWorkPressure:= THIS^.stERParams.rWorkForceB * 1000, 
                                  bPressureRegulation:= TRUE,
                                  eSpeedType:= E_SPEED_TYPE.MM_PER_SECOND, 
                                  rSpeed:= THIS^.stERParams.rSpeedB)
      AND THIS^.itfCounterCyl.M_ToHP( ePressureType:= E_PRESSURE_TYPE.FORCE, 
                                      rWorkPressure:= THIS^.stERParams.rLoadForceB * 1000, 
                                      bPressureRegulation:= TRUE,
                                      eSpeedType:= E_SPEED_TYPE.PERCENT, 
                                      rSpeed:= 100)
			THEN 
        THIS^.stSeqCtrlGeneral.iInternalSeqStateCase := 80;
			END_IF
      
    72: // Move to HP (Min position + 10)
      IF TRUE
      AND THIS^.itfTestCyl.M_ToHP(ePressureType:= E_PRESSURE_TYPE.VALUE, 
                                  rWorkPressure:= 0, 
                                  bPressureRegulation:= FALSE,
                                  eSpeedType:= E_SPEED_TYPE.MM_PER_SECOND, 
                                  rSpeed:= THIS^.stERParams.rSpeedB)
      AND THIS^.itfCounterCyl.M_ToWP( ePressureType:= E_PRESSURE_TYPE.FORCE, 
                                      rWorkPressure:= stERParams.rLoadForceA * 1000, 
                                      bPressureRegulation:= FALSE,
                                      eSpeedType:= E_SPEED_TYPE.PERCENT, 
                                      rSpeed:= 50)
			THEN 
        THIS^.stSeqCtrlGeneral.iInternalSeqStateCase := 80;
			END_IF
      
    80: // Move to WP (Min position + 10)
      IF TRUE
			THEN 
        IF THIS^.itfTestCyl.P_Position <= ABS(THIS^.stERParams.rTurningPointHP) THEN
          THIS^.udiCurrentCycle := THIS^.udiCurrentCycle + 1;
          THIS^.udiERTotalCycles := THIS^.udiERTotalCycles + 1;
				  THIS^.stSeqCtrlGeneral.iInternalSeqStateCase := 15; // Jump backward
        END_IF
			END_IF
      
    1000: // Move to WP (Max position - 10)
      IF TRUE
      AND THIS^.itfTestCyl.M_ToWP(ePressureType:= E_PRESSURE_TYPE.FORCE, 
                                  rWorkPressure:= THIS^.stERParams.rWorkForceA * 1000, 
                                  bPressureRegulation:= TRUE,
                                  eSpeedType:= E_SPEED_TYPE.MM_PER_SECOND, 
                                  rSpeed:= THIS^.stERParams.rSpeedA)
      AND THIS^.itfCounterCyl.M_ToWP( ePressureType:= E_PRESSURE_TYPE.FORCE, 
                                      rWorkPressure:= THIS^.stERParams.rLoadForceA * 1000, 
                                      bPressureRegulation:= TRUE,
                                      eSpeedType:= E_SPEED_TYPE.PERCENT, 
                                      rSpeed:= 50)
			THEN 
        THIS^.stSeqCtrlGeneral.iInternalSeqStateCase := 1010;
			END_IF
      
    1010: // Move to WP (Max position - 10)
      IF TRUE
			THEN 
        IF THIS^.itfTestCyl.P_Position >= THIS^.itfTestCyl.P_StrokeLength / 2 THEN
				  THIS^.stSeqCtrlGeneral.iInternalSeqStateCase := 1020; 
        END_IF
			END_IF
      
    1020: // Exit seq - Stop
      IF TRUE
      AND _m_Delay(DelayTime:= T#1S) 
      AND THIS^.itfTestCyl.M_StopAndLock()
      AND THIS^.itfCounterCyl.M_Stop()
			THEN 
				THIS^.stSeqCtrlGeneral.iInternalSeqStateCase := 1030;
			END_IF
      
    1030: // Exit seq - Disable low pressure circuit
      IF TRUE
      AND _m_Delay(DelayTime:= T#1S)
      AND THIS^.itfCounterCyl.M_LowPressureCircuit(bAdd:= FALSE)
			THEN 
				THIS^.stSeqCtrlGeneral.iInternalSeqStateCase := 1040;
			END_IF 
      
    1040: // Set pressure
      IF TRUE 
			AND THIS^.itfCounterCyl.M_SetWorkPressureZero()
      AND THIS^.itfTestCyl.M_SetWorkPressureZero()
			THEN 
				THIS^.stSeqCtrlGeneral.iInternalSeqStateCase := 1050; 
			END_IF
      
    1050: // Remove pump 2
      IF TRUE 
			AND THIS^.itfTestCyl.M_Pump2Add(bAdd:= FALSE)
			THEN
        THIS^.stSeqCtrlGeneral.iInternalSeqStateCase := 1060; 
			END_IF
      
    1060: // Remove pump 3
      IF TRUE 
			AND THIS^.itfTestCyl.M_Pump3Add(bAdd:= FALSE)
			THEN
        THIS^.stSeqCtrlGeneral.iInternalSeqStateCase := 1070; 
			END_IF
      
    1070: // Remove pump 4
      IF TRUE 
			AND THIS^.itfTestCyl.M_Pump4Add(bAdd:= FALSE)
			THEN
        IF TRUE
        AND (THIS^.stERParams.rSpeedA > THIS^.rMaxSpeedInMmPerSWP * THIS^.rSpeedEfficiencyFactor
        OR THIS^.stERParams.rSpeedB > THIS^.rMaxSpeedInMmPerSHP * THIS^.rSpeedEfficiencyFactor) 
        THEN
          THIS^.stSeqCtrlGeneral.iInternalSeqStateCase := 1080; 
        ELSE
          THIS^.stSeqCtrlGeneral.iInternalSeqStateCase := 9999; 
        END_IF
			END_IF
      
    1080: // Set Pressure to zero
      IF TRUE 
      AND THIS^.itfPump2Pressure.M_SetLimit(ePressureType:= E_PRESSURE_TYPE.PERCENT, rLimit:= 0)
      AND THIS^.itfPump3Pressure.M_SetLimit(ePressureType:= E_PRESSURE_TYPE.PERCENT, rLimit:= 0)
			AND THIS^.itfPump4Pressure.M_SetLimit(ePressureType:= E_PRESSURE_TYPE.PERCENT, rLimit:= 0)
			THEN
        THIS^.stSeqCtrlGeneral.iInternalSeqStateCase := 9999; 
			END_IF
      
	ELSE
		THIS^.stSeqCtrlGeneral.eActiveSeqState := E_SEQ_GENERAL.DONE;  
	END_CASE
	THIS^.stSeqCtrlGeneral.strExtraInfo := CONCAT('Internal state: ', TO_STRING(THIS^.stSeqCtrlGeneral.iInternalSeqStateCase));

E_SEQ_GENERAL.DONE:;
E_SEQ_GENERAL.ERROR:;
E_SEQ_GENERAL.TIME_OUT:; 

IF TRUE
AND THIS^.stSeqCtrlGeneral.bTimeOutActiveQuit 
THEN
  THIS^.stSeqCtrlGeneral.strExtraInfo := 'Bitte quittieren und erneut testen';
  IF TRUE
  //AND itfOpMode.P_QUIT
  THEN
    THIS^.stSeqCtrlGeneral.eActiveSeqState := E_SEQ_GENERAL.EXECUTE;
	END_IF
  
END_IF

ELSE
  THIS^.stSeqCtrlGeneral.eActiveSeqState := E_SEQ_GENERAL.ERROR;
END_CASE
END_METHOD

METHOD PRIVATE _m_Seq_INIT : E_SEQ_PROCESS
VAR_INPUT
END_VAR
VAR
	ActiveSeq: STRING;
END_VAR
VAR
	
END_VAR
//THIS^._m_GeneralStepSetting(StepType:=E_STEP_STATE_TYPE.INIT,
ActiveSeq := TO_STRING(THIS^.eSeq);

CASE THIS^.stSeqCtrlGeneral.eActiveSeqState OF
E_SEQ_GENERAL.READY:;

	
E_SEQ_GENERAL.EXECUTE:;
	IF TRUE
	THEN
		THIS^.stSeqCtrlGeneral.eActiveSeqState := E_SEQ_GENERAL.RESET;
	END_IF
E_SEQ_GENERAL.RESET:;
	stSeqCtrlGeneral.iInternalSeqStateCase := 0;
	IF TRUE
	THEN
    THIS^.udiERTotalCycles := 0;
		THIS^.stSeqCtrlGeneral.eActiveSeqState := E_SEQ_GENERAL.BUSY;
	END_IF
  
E_SEQ_GENERAL.BUSY:;
	CASE THIS^.stSeqCtrlGeneral.iInternalSeqStateCase OF
    0:  // Switch off the counter and test pump
      IF TRUE 
			//AND THIS^.itfCounterCylPump.M_Off()
      //AND THIS^.itfTestCylPump.M_Off()
			THEN 
				THIS^.stSeqCtrlGeneral.iInternalSeqStateCase := 10; 
			END_IF
      
    10: // Enable counter and low pressure pump bypass
      IF TRUE 
			AND THIS^.itfCounterCylPump.M_Bypass(bEnable:= TRUE)
			THEN 
				THIS^.stSeqCtrlGeneral.iInternalSeqStateCase := 20; 
			END_IF
      
    20: // Disable pump 2
      IF TRUE 
			AND THIS^.itfTestCyl.M_Pump2Add(bAdd:= FALSE)
      AND THIS^.itfPump2Pressure.M_SetLimit(ePressureType:= E_PRESSURE_TYPE.PERCENT, rLimit:= 0)
			THEN
        THIS^.stSeqCtrlGeneral.iInternalSeqStateCase := 30; 
			END_IF
      
    30: // Disable pump 3
      IF TRUE 
			AND THIS^.itfTestCyl.M_Pump3Add(bAdd:= FALSE)
      AND THIS^.itfPump3Pressure.M_SetLimit(ePressureType:= E_PRESSURE_TYPE.PERCENT, rLimit:= 0)
			THEN
        THIS^.stSeqCtrlGeneral.iInternalSeqStateCase := 40; 
			END_IF
      
    40: // Disable pump 4
      IF TRUE 
			AND THIS^.itfTestCyl.M_Pump4Add(bAdd:= FALSE)
      AND THIS^.itfPump4Pressure.M_SetLimit(ePressureType:= E_PRESSURE_TYPE.PERCENT, rLimit:= 0)
			THEN
        THIS^.stSeqCtrlGeneral.iInternalSeqStateCase := 50; 
			END_IF
      
		50:	// Reset counter cylinder
      IF TRUE 
			AND THIS^.itfCounterCyl.M_Reset()
			THEN 
				THIS^.stSeqCtrlGeneral.iInternalSeqStateCase := 60; 
			END_IF
      
		60: // Reset test cylinder
      IF TRUE 
			AND THIS^.itfTestCyl.M_Reset()
			THEN 
				THIS^.stSeqCtrlGeneral.iInternalSeqStateCase := 70; 
			END_IF
      
		70: // Turn on the counter, test and low pressure pump
      IF TRUE 
			AND THIS^.itfCounterCylPump.M_On() 
      AND THIS^.itfTestCylPump.M_On()
			THEN 
				THIS^.stSeqCtrlGeneral.iInternalSeqStateCase := 1000; 
			END_IF
      
    1000: // Exit step
      IF TRUE
			THEN 
				THIS^.stSeqCtrlGeneral.iInternalSeqStateCase := 9999;
			END_IF
      
	ELSE
		THIS^.stSeqCtrlGeneral.eActiveSeqState := E_SEQ_GENERAL.DONE;  
	END_CASE
	THIS^.stSeqCtrlGeneral.strExtraInfo := CONCAT('Internal state: ', TO_STRING(THIS^.stSeqCtrlGeneral.iInternalSeqStateCase));
E_SEQ_GENERAL.DONE:;
E_SEQ_GENERAL.ERROR:;
E_SEQ_GENERAL.TIME_OUT:; 

IF TRUE
AND THIS^.stSeqCtrlGeneral.bTimeOutActiveQuit 
THEN
  THIS^.stSeqCtrlGeneral.strExtraInfo := 'Bitte quittieren und erneut testen';
  IF TRUE
  //AND itfOpMode.P_QUIT
  THEN
    THIS^.stSeqCtrlGeneral.eActiveSeqState := E_SEQ_GENERAL.EXECUTE;
	END_IF
  
END_IF

ELSE
  THIS^.stSeqCtrlGeneral.eActiveSeqState := E_SEQ_GENERAL.ERROR;
END_CASE
END_METHOD

METHOD PRIVATE _m_Seq_LEAK_TEST_1 : E_SEQ_PROCESS
VAR_INPUT
END_VAR
VAR
  ActiveSeq: STRING;
END_VAR
//THIS^._m_GeneralStepSetting(StepType:=E_STEP_STATE_TYPE.INIT,
ActiveSeq := TO_STRING(THIS^.eSeq);

// Distance record
_m_DistanceRecord();

CASE THIS^.stSeqCtrlGeneral.eActiveSeqState OF
E_SEQ_GENERAL.READY:;

	
E_SEQ_GENERAL.EXECUTE:;
	IF TRUE
	AND _m_Delay(T#1S)
	THEN
		THIS^.stSeqCtrlGeneral.eActiveSeqState := E_SEQ_GENERAL.RESET;
	END_IF
  
E_SEQ_GENERAL.RESET:;
	stSeqCtrlGeneral.iInternalSeqStateCase := 0;
	IF TRUE
	THEN
		THIS^.stSeqCtrlGeneral.eActiveSeqState := E_SEQ_GENERAL.BUSY;
	END_IF
  
E_SEQ_GENERAL.BUSY:;
	CASE THIS^.stSeqCtrlGeneral.iInternalSeqStateCase OF
		0: // Check if enable
      IF TRUE
      AND THIS^.bEnable 
      THEN
        THIS^.stSeqCtrlGeneral.iInternalSeqStateCase := 10; 
      ELSE
        THIS^.stSeqCtrlGeneral.iInternalSeqStateCase := 9999; 
			END_IF

    10: // Disable low pressure mode and enable bypass to low pressure pump
      IF TRUE 
			AND THIS^.itfTestCyl.M_LowPressureMode(bSet:= FALSE, ePressureType:= E_PRESSURE_TYPE.VALUE, rWorkPressure:= 0)
			THEN 
				THIS^.stSeqCtrlGeneral.iInternalSeqStateCase := 20; 
			END_IF
      
    20: // Shut off low pressure circuit to counter cylinder and switch off pump
      IF TRUE 
			AND THIS^.itfCounterCyl.M_LowPressureCircuit(bAdd:= FALSE)
			THEN 
				THIS^.stSeqCtrlGeneral.iInternalSeqStateCase := 30; 
			END_IF
      
    30: // Disable pump 2
      IF TRUE 
			AND THIS^.itfTestCyl.M_Pump2Add(bAdd:= FALSE)
      //AND THIS^.itfPump2Pressure.M_SetLimit(ePressureType:= E_PRESSURE_TYPE.PERCENT, rLimit:= 0)
			THEN
        THIS^.stSeqCtrlGeneral.iInternalSeqStateCase := 40; 
			END_IF
      
    40: // Disable pump 3
      IF TRUE 
			AND THIS^.itfTestCyl.M_Pump3Add(bAdd:= FALSE)
      //AND THIS^.itfPump3Pressure.M_SetLimit(ePressureType:= E_PRESSURE_TYPE.PERCENT, rLimit:= 0)
			THEN
        THIS^.stSeqCtrlGeneral.iInternalSeqStateCase := 50; 
			END_IF
      
    50: // Disable pump 4
      IF TRUE 
			AND THIS^.itfTestCyl.M_Pump4Add(bAdd:= FALSE)
      //AND THIS^.itfPump4Pressure.M_SetLimit(ePressureType:= E_PRESSURE_TYPE.PERCENT, rLimit:= 0)
			THEN
        IF THIS^.bDoubleActing THEN
          THIS^.stSeqCtrlGeneral.iInternalSeqStateCase := 60; 
        ELSE
          THIS^.stSeqCtrlGeneral.iInternalSeqStateCase := 61; 
        END_IF
			END_IF
        
    60: // Move to HP (Min position + 10mm)
      IF TRUE
      AND THIS^.itfTestCyl.M_ToHP(ePressureType:= E_PRESSURE_TYPE.FORCE, 
                                  rWorkPressure:= THIS^.stLT1Params.rLoadForceB * 1000, 
                                  bPressureRegulation:= FALSE,
                                  eSpeedType:= E_SPEED_TYPE.PERCENT, 
                                  rSpeed:= 50)
      AND THIS^.itfCounterCyl.M_ToHP(ePressureType:= E_PRESSURE_TYPE.VALUE, 
                                     rWorkPressure:= 0, 
                                     bPressureRegulation:= FALSE,
                                     eSpeedType:= E_SPEED_TYPE.PERCENT, 
                                     rSpeed:= 50)
			THEN 
        IF THIS^.itfTestCyl.P_Position <= ABS(THIS^.stLT1Params.rDistanceBeforeEndPosHP) THEN
				  THIS^.stSeqCtrlGeneral.iInternalSeqStateCase := 70; 
        END_IF
			END_IF
      
    61: // Move to HP (Min position + 10mm)
      IF TRUE
      AND THIS^.itfTestCyl.M_ToHP(ePressureType:= E_PRESSURE_TYPE.VALUE, 
                                  rWorkPressure:= 0, 
                                  bPressureRegulation:= FALSE,
                                  eSpeedType:= E_SPEED_TYPE.PERCENT, 
                                  rSpeed:= 50)
      AND THIS^.itfCounterCyl.M_ToWP(ePressureType:= E_PRESSURE_TYPE.FORCE, 
                                     rWorkPressure:= THIS^.stLT1Params.rLoadForceA * 1000, 
                                     bPressureRegulation:= FALSE,
                                     eSpeedType:= E_SPEED_TYPE.PERCENT, 
                                     rSpeed:= 50)
			THEN 
        IF THIS^.itfTestCyl.P_Position <= ABS(THIS^.stLT1Params.rDistanceBeforeEndPosHP) THEN
				  THIS^.stSeqCtrlGeneral.iInternalSeqStateCase := 70; 
        END_IF
			END_IF
      
    70: // Stop and lock
      IF TRUE
      AND _m_Delay(DelayTime:= T#1S)
      AND THIS^.itfTestCyl.M_StopAndLock()
      AND THIS^.itfCounterCyl.M_Stop()
			THEN 
        THIS^.stSeqCtrlGeneral.iInternalSeqStateCase := 80; 
			END_IF
      
    80: // Set cylinder pressure to 0
      IF TRUE
      AND THIS^.itfTestCyl.M_SetWorkPressureZero()
			THEN 
        THIS^.stSeqCtrlGeneral.iInternalSeqStateCase := 90; 
			END_IF
      
    90: // Start leak test push (HP endposition + 10mm)
      IF TRUE
      AND _m_Delay(DelayTime:= T#1S)
      AND THIS^.itfCounterCyl.M_ToWP(ePressureType:= E_PRESSURE_TYPE.FORCE, 
                                     rWorkPressure:= THIS^.stLT1Params.rLoadForceA * 1000, 
                                     bPressureRegulation:= TRUE,
                                     eSpeedType:= E_SPEED_TYPE.PERCENT, 
                                     rSpeed:= 100)
			THEN 
        THIS^.stSeqCtrlGeneral.iInternalSeqStateCase := 100;
			END_IF
      
    100: // Leak detection
      IF TRUE
      AND _m_LeakTest1_LeakDet()
			THEN 
        THIS^.stSeqCtrlGeneral.iInternalSeqStateCase := 110;
			END_IF
      
    110: // Stop and delay
      IF TRUE
      AND _m_Delay(DelayTime:= REAL_TO_TIME(THIS^.stLT1Params.rRestDelay * 1000))
      AND THIS^.itfCounterCyl.M_Stop()
			THEN 
        IF THIS^.bDoubleActing THEN
          THIS^.stSeqCtrlGeneral.iInternalSeqStateCase := 120;
        ELSE
          THIS^.stSeqCtrlGeneral.iInternalSeqStateCase := 150;
        END_IF
			END_IF
      
    120: // Start leak test pull (HP endposition + 10mm)
      IF TRUE
      AND _m_Delay(DelayTime:= T#1S)
      AND THIS^.itfCounterCyl.M_ToHP(ePressureType:= E_PRESSURE_TYPE.FORCE, 
                                     rWorkPressure:= THIS^.stLT1Params.rLoadForceB * 1000, 
                                     bPressureRegulation:= TRUE,
                                     eSpeedType:= E_SPEED_TYPE.PERCENT, 
                                     rSpeed:= 100)
			THEN 
        THIS^.stSeqCtrlGeneral.iInternalSeqStateCase := 130;
			END_IF
      
    130: // Leak detection
      IF TRUE
      AND _m_LeakTest1_LeakDet()
			THEN 
        THIS^.stSeqCtrlGeneral.iInternalSeqStateCase := 140;
			END_IF
      
    140: // Stop and delay
      IF TRUE
      AND _m_Delay(DelayTime:= REAL_TO_TIME(THIS^.stLT1Params.rRestDelay))
      AND THIS^.itfCounterCyl.M_Stop()
			THEN 
        THIS^.stSeqCtrlGeneral.iInternalSeqStateCase := 150;
			END_IF
      
    150: // Move to WP (Max position - 10mm)
      IF TRUE
      AND THIS^.itfTestCyl.M_ToWP(ePressureType:= E_PRESSURE_TYPE.FORCE, 
                                  rWorkPressure:= THIS^.stLT1Params.rLoadForceA * 1000, 
                                  bPressureRegulation:= FALSE,
                                  eSpeedType:= E_SPEED_TYPE.PERCENT, 
                                  rSpeed:= 50)
      AND THIS^.itfCounterCyl.M_ToWP(ePressureType:= E_PRESSURE_TYPE.VALUE, 
                                     rWorkPressure:= 0, 
                                     bPressureRegulation:= FALSE,
                                     eSpeedType:= E_SPEED_TYPE.PERCENT, 
                                     rSpeed:= 50)
			THEN 
        IF THIS^.itfTestCyl.P_Position >= THIS^.itfTestCyl.P_StrokeLength - ABS(THIS^.stLT1Params.rDistanceBeforeEndPosWP) THEN
				  THIS^.stSeqCtrlGeneral.iInternalSeqStateCase := 160; 
        END_IF
			END_IF
      
    160: // Stop and lock
      IF TRUE
      AND _m_Delay(DelayTime:= T#1S)
      AND THIS^.itfTestCyl.M_StopAndLock()
      AND THIS^.itfCounterCyl.M_Stop()
			THEN 
        THIS^.stSeqCtrlGeneral.iInternalSeqStateCase := 170; 
			END_IF
      
    170: // Set cylinder pressure to 0
      IF TRUE
      AND THIS^.itfTestCyl.M_SetWorkPressureZero()
			THEN 
        THIS^.stSeqCtrlGeneral.iInternalSeqStateCase := 180; 
			END_IF
      
    180: // Start leak test push (WP endposition - 10mm)
      IF TRUE
      AND _m_Delay(DelayTime:= T#1S)
      AND THIS^.itfCounterCyl.M_ToWP(ePressureType:= E_PRESSURE_TYPE.FORCE, 
                                     rWorkPressure:= THIS^.stLT1Params.rLoadForceA * 1000, 
                                     bPressureRegulation:= TRUE,
                                     eSpeedType:= E_SPEED_TYPE.PERCENT, 
                                     rSpeed:= 100)
			THEN 
        THIS^.stSeqCtrlGeneral.iInternalSeqStateCase := 190;
			END_IF
      
    190: // Leak detection
      IF TRUE
      AND _m_LeakTest1_LeakDet()
			THEN 
        THIS^.stSeqCtrlGeneral.iInternalSeqStateCase := 200;
			END_IF
      
    200: // Stop and delay
      IF TRUE
      AND _m_Delay(DelayTime:= REAL_TO_TIME(THIS^.stLT1Params.rRestDelay * 1000))
      AND THIS^.itfCounterCyl.M_Stop()
			THEN 
        IF THIS^.bDoubleActing THEN
          THIS^.stSeqCtrlGeneral.iInternalSeqStateCase := 210; 
        ELSE
          THIS^.stSeqCtrlGeneral.iInternalSeqStateCase := 241; 
        END_IF
			END_IF
      
    210: // Start leak test pull (WP endposition - 10mm)
      IF TRUE
      AND _m_Delay(DelayTime:= T#1S)
      AND THIS^.itfCounterCyl.M_ToHP(ePressureType:= E_PRESSURE_TYPE.FORCE, 
                                     rWorkPressure:= THIS^.stLT1Params.rLoadForceB * 1000, 
                                     bPressureRegulation:= TRUE,
                                     eSpeedType:= E_SPEED_TYPE.PERCENT, 
                                     rSpeed:= 100)
			THEN 
        THIS^.stSeqCtrlGeneral.iInternalSeqStateCase := 220;
			END_IF
      
